// SIMATIC STEP 7 (V5.x) project Project
// CPU: CPU 315-2 DP
// station: Hardware
// station: SIMATIC 300(1)
// station: _S7H_BUSSYSTEM_CT
// station: P_ADR_BUS
// program: S7 Program(1)

SYMBOL_TABLE
"GLV"	DB 1	DB 1
"A_Sensors"	DB 2	DB 2
"DI"	DB 3	DB 3
"SensorsSettings"	DB 4	DB 4
"Valves"	DB 5	DB 5
"BD_Coils"	DB 6	DB 6
"KB1_1_Coils"	DB 7	DB 7
"KB1_2_Coils"	DB 8	DB 8
"KB2_Coils"	DB 9	DB 9
"PO1_1_Coils"	DB 10	DB 10
"PO1_2_Coils"	DB 11	DB 11
"GA1_1_Coils"	DB 12	DB 12
"GA1_2_Coils"	DB 13	DB 13
"GA2_1_Coils"	DB 14	DB 14
"GA2_2_Coils"	DB 15	DB 15
"BD_AI_1"	DB 16	DB 16
"KB1_1_AI_1"	DB 17	DB 17
"KB1_1_AI_2"	DB 18	DB 18
"KB1_1_AI_3"	DB 19	DB 19
"KB1_2_AI_1"	DB 20	DB 20
"KB1_2_AI_2"	DB 21	DB 21
"KB1_2_AI_3"	DB 22	DB 22
"KB2_AI_1"	DB 23	DB 23
"KB2_AI_2"	DB 24	DB 24
"KB2_AI_3"	DB 25	DB 25
"KB2_AI_4"	DB 26	DB 26
"PO1_1_AI"	DB 27	DB 27
"PO1_2_AI"	DB 28	DB 28
"GA1_1_AI_1"	DB 29	DB 29
"GA1_1_AI_2"	DB 30	DB 30
"GA1_2_AI_1"	DB 31	DB 31
"GA1_2_AI_2"	DB 32	DB 32
"GA2_1_AI_1"	DB 33	DB 33
"GA2_1_AI_2"	DB 34	DB 34
"KD1_1_AI"	DB 35	DB 35
"GA2_2_AI_1"	DB 36	DB 36
"GA2_2_AI_2"	DB 37	DB 37
"KD1_1_AI_2"	DB 38	DB 38
"KD1_1_AI_3"	DB 39	DB 39
"KD1_1_AI_4"	DB 40	DB 40
"KD1_1_AI_5"	DB 41	DB 41
"KD1_1_Coils"	DB 42	DB 42
"BD1_ARR_AI"	DB 43	DB 43
"BD_AI_2"	DB 44	DB 44
"BD_AI_3"	DB 45	DB 45
"BD_DO_1"	DB 46	DB 46
"BD_DO_2"	DB 47	DB 47
"GA1_1_DO"	DB 48	DB 48
"GA1_2_DO"	DB 49	DB 49
"GA2_1_DO"	DB 50	DB 50
"GA2_2_DO"	DB 51	DB 51
"BD_REAL"	DB 52	DB 52
"KB1_1_REAL"	DB 53	DB 53
"KB1_2_REAL"	DB 54	DB 54
"KB2_REAL"	DB 55	DB 55
"PO1_1_REAL"	DB 56	DB 56
"PO1_2_REAL"	DB 57	DB 57
"GA1_1_REAL"	DB 58	DB 58
"GA1_2_REAL"	DB 59	DB 59
"GA2_1_REAL"	DB 60	DB 60
"GA2_2_REAL"	DB 61	DB 61
"KD_REAL"	DB 62	DB 62
"ModbusVars"	DB 63	DB 63
"BD_Outputs_1"	DB 64	DB 64
"BD_Outputs_2"	DB 65	DB 65
"PO1_1_Outputs"	DB 66	DB 66
"PO1_2_Outputs"	DB 67	DB 67
"GA1_1_Outputs"	DB 68	DB 68
"GA1_2_Outputs"	DB 69	DB 69
"GA2_1_Outputs"	DB 97	DB 97
"GA2_2_Outputs"	DB 98	DB 98
"BD_OutputBytes_1"	DB 99	DB 99
"BD_OutputBytes_2"	DB 111	DB 111
"PO1_1_OutBytes"	DB 112	DB 112
"PO1_2_OutBytes"	DB 113	DB 113
"GA1_1_OutBytes"	DB 114	DB 114
"GA1_2_OutBytes"	DB 115	DB 115
"GA2_1_OutBytes"	DB 116	DB 116
"GA2_2_OutBytes"	DB 117	DB 117
"StartStop"	DB 118	DB 118
"StartStopBytes"	DB 119	DB 119
"KB2_AI_Bearer"	DB 128	DB 128
"KB2_AI_Vibration"	DB 129	DB 129
"ModbusAddresses"	DB 130	DB 130
"PO2_AI"	DB 131	DB 131
"PO2_Reals"	DB 132	DB 132
"PO2_AI2"	DB 133	DB 133
"DI_Bytes"	DB 134	DB 134
"PCV10_PID_Vars"	DB 135	DB 135
"PCV21_PID_Vars"	DB 136	DB 136
"PCV22_PID_Vars"	DB 137	DB 137
"PCV25_PID_Vars"	DB 138	DB 138
"ValvesVars"	DB 139	DB 139
"SensorsAlarmSettings"	DB 140	DB 140
"BD_MaxMin"	DB 141	DB 141
"GA1_1_MinMax"	DB 142	DB 142
"GA1_2_MinMax"	DB 143	DB 143
"GA2_1_MinMax"	DB 144	DB 144
"GA2_2_MinMax"	DB 145	DB 145
"KB1_1_MinMax"	DB 146	DB 146
"KB1_2_MinMax"	DB 147	DB 147
"KD2_ManMax"	DB 148	DB 148
"PO1_1_MaxMin"	DB 149	DB 149
"PO1_2_MinMax"	DB 150	DB 150
"ProcessSettings"	DB 151	DB 151
"ProcessVars"	DB 152	DB 152
"PrepareStartStop"	DB 153	DB 153
"PO2_Coils"	DB 154	DB 154
"PO2_MinMax"	DB 155	DB 155
"ZB1"	DB 777	FB 38
"ZB2"	DB 778	FB 38
"ZB3"	DB 779	FB 38
"ZB4"	DB 780	FB 38
"ValvesPrgDB"	DB 781	FB 39
"BD_GetReals"	FB 1	FB 1
"KB1_1_GetReals"	FB 2	FB 2
"KB1_2_GetReals"	FB 3	FB 3
"KB2_GetReals"	FB 4	FB 4
"PO1_1_GetReals"	FB 5	FB 5
"PO1_2_GetReals"	FB 6	FB 6
"P_RCV_RK"	FB 7	FB 7	// Receive Data / Provide Data
"P_SND_RK"	FB 8	FB 8	// Send Data / Fetch Data
"GA1_1_GetReal"	FB 9	FB 9
"MBMAREQ"	FB 10	FB 10	// MBMAREQ MODBUS MASTER REQUEST FUNCTION BLOCK
"GA1_2_GetReals"	FB 11	FB 11
"GA2_1_GetReals"	FB 12	FB 12
"GA2_2_GetReals"	FB 13	FB 13
"KD_GetReals"	FB 14	FB 14
"ModbusReal"	FB 15	FB 15
"ModbusCoils"	FB 16	FB 16
"ModbusOutputs"	FB 17	FB 17
"BD_GetOutputs"	FB 18	FB 18
"PO1_1_GetOutputs"	FB 19	FB 19
"PO1_2_GetOutputs"	FB 20	FB 20
"GA1_1_GetOutputs"	FB 21	FB 21
"GA1_2_GetOutputs"	FB 22	FB 22
"GA2_1_GetOutputs"	FB 23	FB 23
"GA2_2_GetOutputs"	FB 24	FB 24
"ModbusStartStop"	FB 25	FB 25
"GetStartStopBytes"	FB 26	FB 26
"GetAll"	FB 27	FB 27
"ModbusAll"	FB 28	FB 28
"InToVars"	FB 29	FB 29
"InToVarsST"	FB 30	FB 30
"PO2_GetReals"	FB 31	FB 31
"DI_ToVars"	FB 32	FB 32
"Valve_PID"	FB 33	FB 33
"fbPID"	FB 34	FB 34
"MBMA341"	FB 35	FB 35	// MBMA341 MODBUS MASTER COMMUNICATION FUNCTION BLOCK
"DERIVATIVE"	FB 36	FB 36
"INTEGRAL"	FB 37	FB 37
"DO_Valve"	FB 38	FB 38
"ValvesPrg"	FB 39	FB 39
"fbProcess_1"	FB 40	FB 40
"CONT_C"	FB 41	FB 41	// Continuous Control
"CONT_S"	FB 42	FB 42	// Step Control
"fbImpulsValve"	FB 43	FB 43
"fbImpulsValveSCL"	FB 44	FB 44
"prProcess"	FB 45	FB 45
"fbPO"	FB 46	FB 46
"fbKB"	FB 47	FB 47
"fbKZA"	FB 48	FB 48
"prDevices"	FB 49	FB 49
"GetCoils"	FB 50	FB 50
"LinTrafo"	FC 1	FC 1
"fnWordPack"	FC 2	FC 2
"fnBytesToReal"	FC 3	FC 3
"fnBytesToRealOneComma"	FC 4	FC 4
"fnBytesToRealPressure"	FC 5	FC 5
"fnBytesToRealTwoComas"	FC 6	FC 6
"StartStopByte"	FC 7	FC 7
"LinTrafoInt"	FC 8	FC 8
"ByteToByte"	FC 9	FC 9
"_DI_XL1_QL3"	I 0.0	BOOL
"_DI_XL2_QL3"	I 0.1	BOOL
"_DI_Q3_Bad"	I 0.2	BOOL
"_DI_AB1_Working"	I 0.3	BOOL
"_DI_Kb_1_1_Working"	I 0.4	BOOL
"_DI_Kb_1_1_Alm"	I 0.5	BOOL
"_DI_Kb_1_2_Working"	I 0.6	BOOL
"_DI_Kb_1_2_Alm"	I 0.7	BOOL
"_DI_Kb_2_Working"	I 1.0	BOOL
"_DI_Kb_2_Alm"	I 1.1	BOOL
"_DI_Kd_1_Working"	I 1.2	BOOL
"_DI_Kd_1_Alm"	I 1.3	BOOL
"_DI_ZB_1_Opn"	I 1.4	BOOL
"_DI_ZB_1_Cls"	I 1.5	BOOL
"_DI_ZB_1_Local"	I 1.6	BOOL
"_DI_ZB_1_Alm"	I 1.7	BOOL
"_DI_ZB_2_Opn"	I 2.0	BOOL
"_DI_ZB_2_Cls"	I 2.1	BOOL
"_DI_ZB_2_Local"	I 2.2	BOOL
"_DI_ZB_2_Alm"	I 2.3	BOOL
"_DI_ZB_3_Opn"	I 2.4	BOOL
"_DI_ZB_3_Cls"	I 2.5	BOOL
"_DI_ZB_3_Local"	I 2.6	BOOL
"_DI_ZB_3_Alm"	I 2.7	BOOL
"_DI_EUV_001_Opn"	I 3.0	BOOL
"_DI_EUV_001_Cls"	I 3.1	BOOL
"_DI_EUV_001_Local"	I 3.2	BOOL
"_DI_EUV_001_Alm"	I 3.3	BOOL
"_DI_EUV_002_Opn"	I 3.4	BOOL
"_DI_EUV_002_Cls"	I 3.5	BOOL
"_DI_EUV_002_Local"	I 3.6	BOOL
"_DI_EUV_002_Alm"	I 3.7	BOOL
"_DI_EUV_003_Opn"	I 4.0	BOOL
"_DI_EUV_003_Cls"	I 4.1	BOOL
"_DI_EUV_003_Local"	I 4.2	BOOL
"_DI_EUV_003_Alm"	I 4.3	BOOL
"QSA_19_1_1"	I 4.4	BOOL
"QSA_23_1_1"	I 4.5	BOOL
"QSA_19_1_2"	I 4.6	BOOL
"QSA_23_1_2"	I 4.7	BOOL
"QSA_19_1_3"	I 5.0	BOOL
"QSA_23_1_3"	I 5.1	BOOL
"QSA_19_1_4"	I 5.2	BOOL
"QSA_23_1_4"	I 5.3	BOOL
"QSA_19_1_5"	I 5.4	BOOL
"QSA_23_1_5"	I 5.5	BOOL
"Q3_BAD"	I 5.6	BOOL
"AB_1_Alm"	I 5.7	BOOL
"AB_2_Working"	I 6.0	BOOL
"AB_2_Alm"	I 6.1	BOOL
"AB_3_Working"	I 6.2	BOOL
"AB_3_Alm"	I 6.3	BOOL
"AB_4_Working"	I 6.4	BOOL
"AB_4_Alm"	I 6.5	BOOL
"P2_Alm"	I 6.6	BOOL
"P2_Working"	I 6.7	BOOL
"P3_Alm"	I 7.0	BOOL
"P3_Working"	I 7.1	BOOL
"IBP_1_Working"	I 7.2	BOOL
"IBP_1_Alm"	I 7.3	BOOL
"IBP_1_Bypas"	I 7.4	BOOL
"IBP_2_Working"	I 7.5	BOOL
"IBP_2_Alm"	I 7.6	BOOL
"IBP_2_Bypas"	I 7.7	BOOL
"_DI_ZB_4_Opn"	I 8.0	BOOL
"_DI_ZB_4_Cls"	I 8.1	BOOL
"_DI_ZB_4_Local"	I 8.2	BOOL
"_DI_ZB_4_Alm"	I 8.3	BOOL
"_KB_1_1_1PIR7"	IW 256	WORD
"_KB_1_2_2PIR7"	IW 258	WORD
"_1PIR6"	IW 260	WORD
"_KZA_1_2_2PIR6"	IW 262	WORD
"_KB_2_PIR8"	IW 264	WORD
"_1PIR20"	IW 266	WORD
"_2PIR20"	IW 268	WORD
"_TIR10"	IW 270	WORD
"_FIR10"	IW 272	WORD
"_PIR5"	IW 274	WORD
"_FIR5"	IW 276	WORD
"_PIRC21"	IW 278	WORD
"_1PIR27"	IW 280	WORD
"_QIRAH3"	IW 282	WORD
"_2PIR27"	IW 284	WORD
"_PIR4"	IW 286	WORD
"_FIR_4"	IW 288	WORD
"_PIRC22"	IW 290	WORD
"_PIRC23"	IW 292	WORD
"_PIRC24"	IW 294	WORD
"_PIRC25"	IW 296	WORD
"_FIR_25"	IW 298	WORD
"_1PIRC26"	IW 300	WORD
"_2PIRC26"	IW 302	WORD
"_C10"	IW 304	WORD
"_TIR5"	IW 306	WORD
"_TIR4"	IW 308	WORD
"_TIR25"	IW 310	WORD
"_AIR1"	IW 312	WORD
"_QIRAH4Q4"	IW 314	WORD
"CYC_INT5"	OB 35	OB 35	// Cyclic Interrupt 5
"_DO_HS1Q1_Acknow"	Q 0.0	BOOL
"_DO_HS1Q1_Check"	Q 0.1	BOOL
"_DO_KB_1_1_Stop"	Q 0.2	BOOL
"_DO_KB_1_1_Start"	Q 0.3	BOOL
"_DO_KB_1_2_Stop"	Q 0.4	BOOL
"_DO_KB_1_2_Start"	Q 0.5	BOOL
"_DO_KB_2_Stop"	Q 0.6	BOOL
"_DO_KB_2_Start"	Q 0.7	BOOL
"_DO_KD_1_Start"	Q 1.0	BOOL
"_DO_KD_1_Stop"	Q 1.1	BOOL
"_DO_ZB_1_CmdOpn"	Q 1.2	BOOL
"_DO_ZB_1_CmdCls"	Q 1.3	BOOL
"_DO_ZB_1_CmdStop"	Q 1.4	BOOL
"_DO_ZB_2_CmdOpn"	Q 1.5	BOOL
"_DO_ZB_2_CmdCls"	Q 1.6	BOOL
"_DO_ZB_2_CmdStop"	Q 1.7	BOOL
"_DO_ZB_3_CmdOpn"	Q 2.0	BOOL
"_DO_ZB_3_CmdCls"	Q 2.1	BOOL
"_DO_ZB_3_CmdStop"	Q 2.2	BOOL
"_DO_AlnVent"	Q 2.3	BOOL
"_DO_ZB_4_CmdOpn"	Q 2.4	BOOL
"_DO_ZB_4_CmdCls"	Q 2.5	BOOL
"_DO_ZB_4_CmdStop"	Q 2.6	BOOL
"_AO_N_Set_PCV10"	QW 256	WORD
"_AO_N_Set_PCV21"	QW 258	WORD
"_AO_Air_Set_PCV22"	QW 260	WORD
"_AO_Air_Set_PCV25"	QW 262	WORD
"RDREC"	SFB 52	SFB 52	// Read a Process Data Record
"WRREC"	SFB 53	SFB 53	// Write a Process Data Record
"DI_Vars"	VAT 1	
"DO_Vars"	VAT 2	
"AI_Vars"	VAT 3	
"AO_Vars"	VAT 4	
END_SYMBOL_TABLE

FUNCTION_BLOCK "BD_GetReals"	// FB 1
VERSION : 0.1
BEGIN
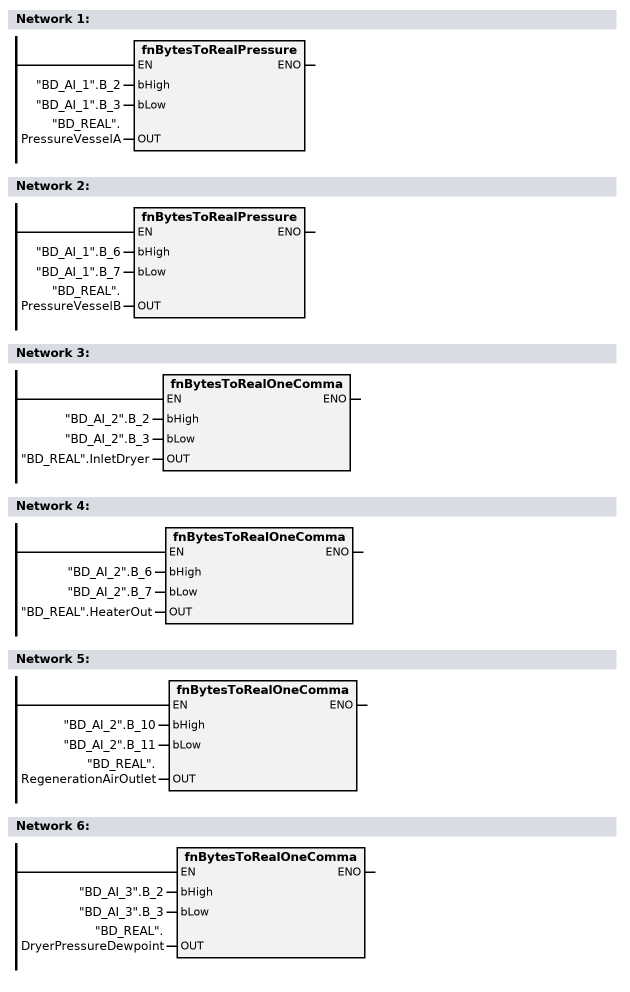
NETWORK
TITLE =
      CALL  "fnBytesToRealPressure" (
           bHigh                    := "BD_AI_1".B_2,
           bLow                     := "BD_AI_1".B_3,
           OUT                      := "BD_REAL".PressureVesselA);
      NOP   0;
NETWORK
TITLE =
      CALL  "fnBytesToRealPressure" (
           bHigh                    := "BD_AI_1".B_6,
           bLow                     := "BD_AI_1".B_7,
           OUT                      := "BD_REAL".PressureVesselB);
      NOP   0;
NETWORK
TITLE =
      CALL  "fnBytesToRealOneComma" (
           bHigh                    := "BD_AI_2".B_2,
           bLow                     := "BD_AI_2".B_3,
           OUT                      := "BD_REAL".InletDryer);
      NOP   0;
NETWORK
TITLE =
      CALL  "fnBytesToRealOneComma" (
           bHigh                    := "BD_AI_2".B_6,
           bLow                     := "BD_AI_2".B_7,
           OUT                      := "BD_REAL".HeaterOut);
      NOP   0;
NETWORK
TITLE =
      CALL  "fnBytesToRealOneComma" (
           bHigh                    := "BD_AI_2".B_10,
           bLow                     := "BD_AI_2".B_11,
           OUT                      := "BD_REAL".RegenerationAirOutlet);
      NOP   0;
NETWORK
TITLE =
      CALL  "fnBytesToRealOneComma" (
           bHigh                    := "BD_AI_3".B_2,
           bLow                     := "BD_AI_3".B_3,
           OUT                      := "BD_REAL".DryerPressureDewpoint);
      NOP   0;
END_FUNCTION_BLOCK

FUNCTION_BLOCK "KB1_1_GetReals"	// FB 2
VERSION : 0.1
BEGIN
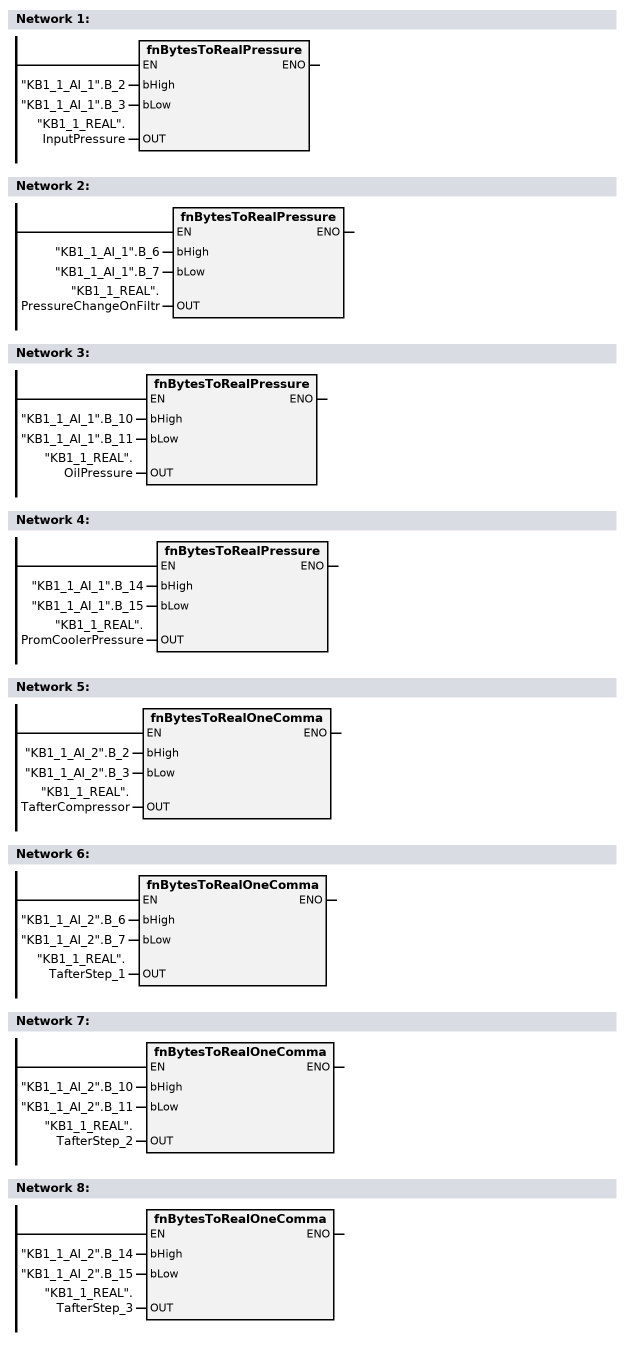
NETWORK
TITLE =
      CALL  "fnBytesToRealPressure" (
           bHigh                    := "KB1_1_AI_1".B_2,
           bLow                     := "KB1_1_AI_1".B_3,
           OUT                      := "KB1_1_REAL".InputPressure);
      NOP   0;
NETWORK
TITLE =
      CALL  "fnBytesToRealPressure" (
           bHigh                    := "KB1_1_AI_1".B_6,
           bLow                     := "KB1_1_AI_1".B_7,
           OUT                      := "KB1_1_REAL".PressureChangeOnFiltr);
      NOP   0;
NETWORK
TITLE =
      CALL  "fnBytesToRealPressure" (
           bHigh                    := "KB1_1_AI_1".B_10,
           bLow                     := "KB1_1_AI_1".B_11,
           OUT                      := "KB1_1_REAL".OilPressure);
      NOP   0;
NETWORK
TITLE =
      CALL  "fnBytesToRealPressure" (
           bHigh                    := "KB1_1_AI_1".B_14,
           bLow                     := "KB1_1_AI_1".B_15,
           OUT                      := "KB1_1_REAL".PromCoolerPressure);
      NOP   0;
NETWORK
TITLE =
      CALL  "fnBytesToRealOneComma" (
           bHigh                    := "KB1_1_AI_2".B_2,
           bLow                     := "KB1_1_AI_2".B_3,
           OUT                      := "KB1_1_REAL".TafterCompressor);
      NOP   0;
NETWORK
TITLE =
      CALL  "fnBytesToRealOneComma" (
           bHigh                    := "KB1_1_AI_2".B_6,
           bLow                     := "KB1_1_AI_2".B_7,
           OUT                      := "KB1_1_REAL".TafterStep_1);
      NOP   0;
NETWORK
TITLE =
      CALL  "fnBytesToRealOneComma" (
           bHigh                    := "KB1_1_AI_2".B_10,
           bLow                     := "KB1_1_AI_2".B_11,
           OUT                      := "KB1_1_REAL".TafterStep_2);
      NOP   0;
NETWORK
TITLE =
      CALL  "fnBytesToRealOneComma" (
           bHigh                    := "KB1_1_AI_2".B_14,
           bLow                     := "KB1_1_AI_2".B_15,
           OUT                      := "KB1_1_REAL".TafterStep_3);
      NOP   0;
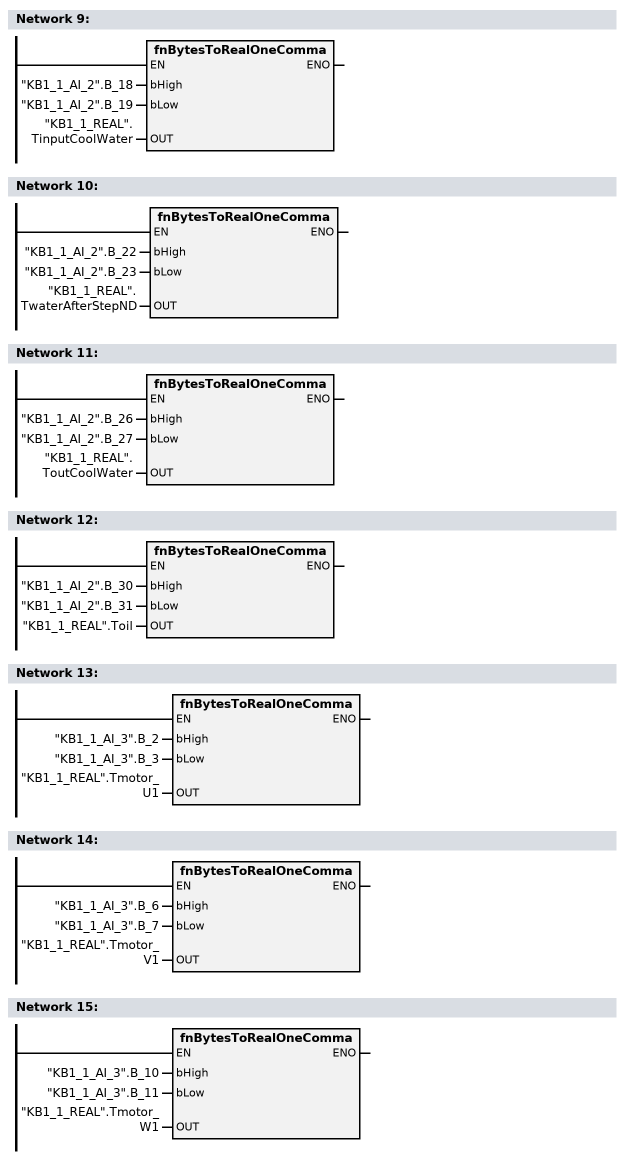
NETWORK
TITLE =
      CALL  "fnBytesToRealOneComma" (
           bHigh                    := "KB1_1_AI_2".B_18,
           bLow                     := "KB1_1_AI_2".B_19,
           OUT                      := "KB1_1_REAL".TinputCoolWater);
      NOP   0;
NETWORK
TITLE =
      CALL  "fnBytesToRealOneComma" (
           bHigh                    := "KB1_1_AI_2".B_22,
           bLow                     := "KB1_1_AI_2".B_23,
           OUT                      := "KB1_1_REAL".TwaterAfterStepND);
      NOP   0;
NETWORK
TITLE =
      CALL  "fnBytesToRealOneComma" (
           bHigh                    := "KB1_1_AI_2".B_26,
           bLow                     := "KB1_1_AI_2".B_27,
           OUT                      := "KB1_1_REAL".ToutCoolWater);
      NOP   0;
NETWORK
TITLE =
      CALL  "fnBytesToRealOneComma" (
           bHigh                    := "KB1_1_AI_2".B_30,
           bLow                     := "KB1_1_AI_2".B_31,
           OUT                      := "KB1_1_REAL".Toil);
      NOP   0;
NETWORK
TITLE =
      CALL  "fnBytesToRealOneComma" (
           bHigh                    := "KB1_1_AI_3".B_2,
           bLow                     := "KB1_1_AI_3".B_3,
           OUT                      := "KB1_1_REAL".Tmotor_U1);
      NOP   0;
NETWORK
TITLE =
      CALL  "fnBytesToRealOneComma" (
           bHigh                    := "KB1_1_AI_3".B_6,
           bLow                     := "KB1_1_AI_3".B_7,
           OUT                      := "KB1_1_REAL".Tmotor_V1);
      NOP   0;
NETWORK
TITLE =
      CALL  "fnBytesToRealOneComma" (
           bHigh                    := "KB1_1_AI_3".B_10,
           bLow                     := "KB1_1_AI_3".B_11,
           OUT                      := "KB1_1_REAL".Tmotor_W1);
      NOP   0;
END_FUNCTION_BLOCK

FUNCTION_BLOCK "KB1_2_GetReals"	// FB 3
VERSION : 0.1
BEGIN
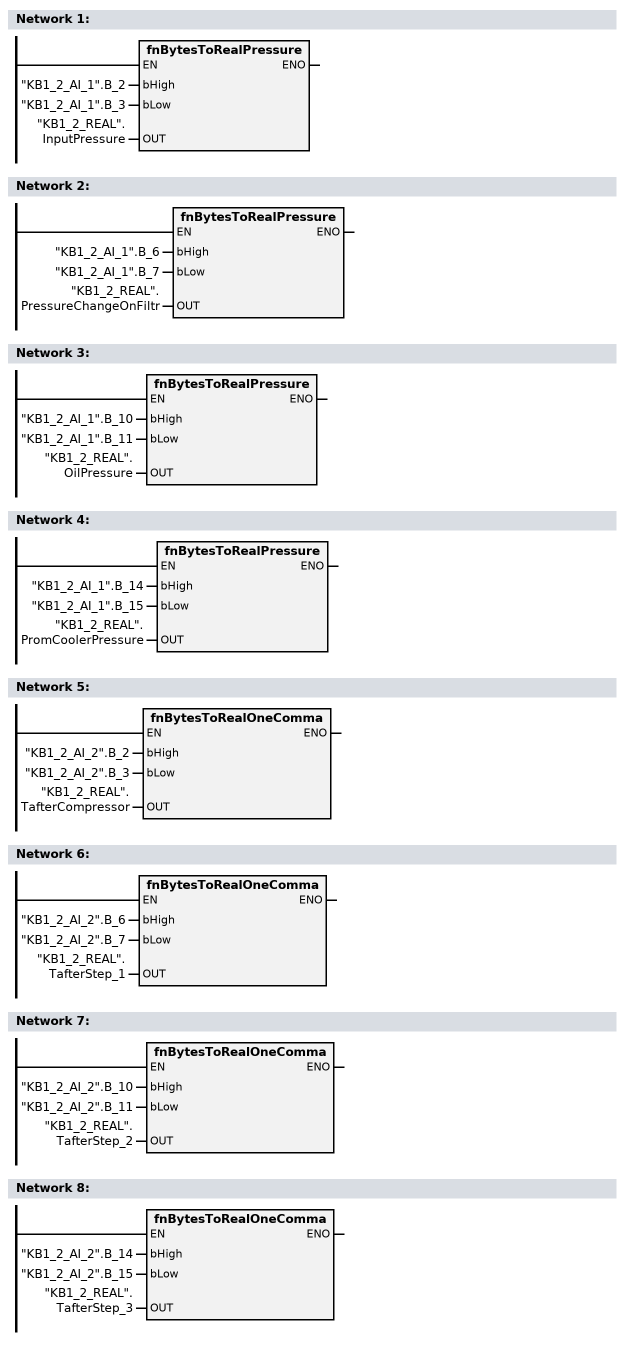
NETWORK
TITLE =
      CALL  "fnBytesToRealPressure" (
           bHigh                    := "KB1_2_AI_1".B_2,
           bLow                     := "KB1_2_AI_1".B_3,
           OUT                      := "KB1_2_REAL".InputPressure);
      NOP   0;
NETWORK
TITLE =
      CALL  "fnBytesToRealPressure" (
           bHigh                    := "KB1_2_AI_1".B_6,
           bLow                     := "KB1_2_AI_1".B_7,
           OUT                      := "KB1_2_REAL".PressureChangeOnFiltr);
      NOP   0;
NETWORK
TITLE =
      CALL  "fnBytesToRealPressure" (
           bHigh                    := "KB1_2_AI_1".B_10,
           bLow                     := "KB1_2_AI_1".B_11,
           OUT                      := "KB1_2_REAL".OilPressure);
      NOP   0;
NETWORK
TITLE =
      CALL  "fnBytesToRealPressure" (
           bHigh                    := "KB1_2_AI_1".B_14,
           bLow                     := "KB1_2_AI_1".B_15,
           OUT                      := "KB1_2_REAL".PromCoolerPressure);
      NOP   0;
NETWORK
TITLE =
      CALL  "fnBytesToRealOneComma" (
           bHigh                    := "KB1_2_AI_2".B_2,
           bLow                     := "KB1_2_AI_2".B_3,
           OUT                      := "KB1_2_REAL".TafterCompressor);
      NOP   0;
NETWORK
TITLE =
      CALL  "fnBytesToRealOneComma" (
           bHigh                    := "KB1_2_AI_2".B_6,
           bLow                     := "KB1_2_AI_2".B_7,
           OUT                      := "KB1_2_REAL".TafterStep_1);
      NOP   0;
NETWORK
TITLE =
      CALL  "fnBytesToRealOneComma" (
           bHigh                    := "KB1_2_AI_2".B_10,
           bLow                     := "KB1_2_AI_2".B_11,
           OUT                      := "KB1_2_REAL".TafterStep_2);
      NOP   0;
NETWORK
TITLE =
      CALL  "fnBytesToRealOneComma" (
           bHigh                    := "KB1_2_AI_2".B_14,
           bLow                     := "KB1_2_AI_2".B_15,
           OUT                      := "KB1_2_REAL".TafterStep_3);
      NOP   0;
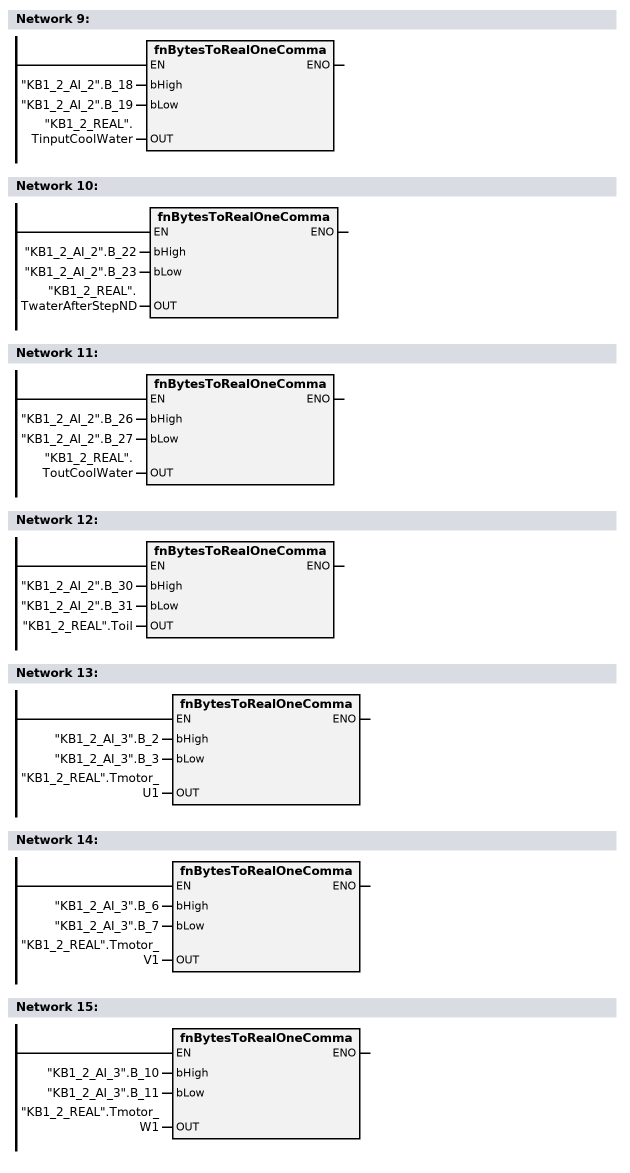
NETWORK
TITLE =
      CALL  "fnBytesToRealOneComma" (
           bHigh                    := "KB1_2_AI_2".B_18,
           bLow                     := "KB1_2_AI_2".B_19,
           OUT                      := "KB1_2_REAL".TinputCoolWater);
      NOP   0;
NETWORK
TITLE =
      CALL  "fnBytesToRealOneComma" (
           bHigh                    := "KB1_2_AI_2".B_22,
           bLow                     := "KB1_2_AI_2".B_23,
           OUT                      := "KB1_2_REAL".TwaterAfterStepND);
      NOP   0;
NETWORK
TITLE =
      CALL  "fnBytesToRealOneComma" (
           bHigh                    := "KB1_2_AI_2".B_26,
           bLow                     := "KB1_2_AI_2".B_27,
           OUT                      := "KB1_2_REAL".ToutCoolWater);
      NOP   0;
NETWORK
TITLE =
      CALL  "fnBytesToRealOneComma" (
           bHigh                    := "KB1_2_AI_2".B_30,
           bLow                     := "KB1_2_AI_2".B_31,
           OUT                      := "KB1_2_REAL".Toil);
      NOP   0;
NETWORK
TITLE =
      CALL  "fnBytesToRealOneComma" (
           bHigh                    := "KB1_2_AI_3".B_2,
           bLow                     := "KB1_2_AI_3".B_3,
           OUT                      := "KB1_2_REAL".Tmotor_U1);
      NOP   0;
NETWORK
TITLE =
      CALL  "fnBytesToRealOneComma" (
           bHigh                    := "KB1_2_AI_3".B_6,
           bLow                     := "KB1_2_AI_3".B_7,
           OUT                      := "KB1_2_REAL".Tmotor_V1);
      NOP   0;
NETWORK
TITLE =
      CALL  "fnBytesToRealOneComma" (
           bHigh                    := "KB1_2_AI_3".B_10,
           bLow                     := "KB1_2_AI_3".B_11,
           OUT                      := "KB1_2_REAL".Tmotor_W1);
      NOP   0;
END_FUNCTION_BLOCK

FUNCTION_BLOCK "KB2_GetReals"	// FB 4
VERSION : 0.1
BEGIN
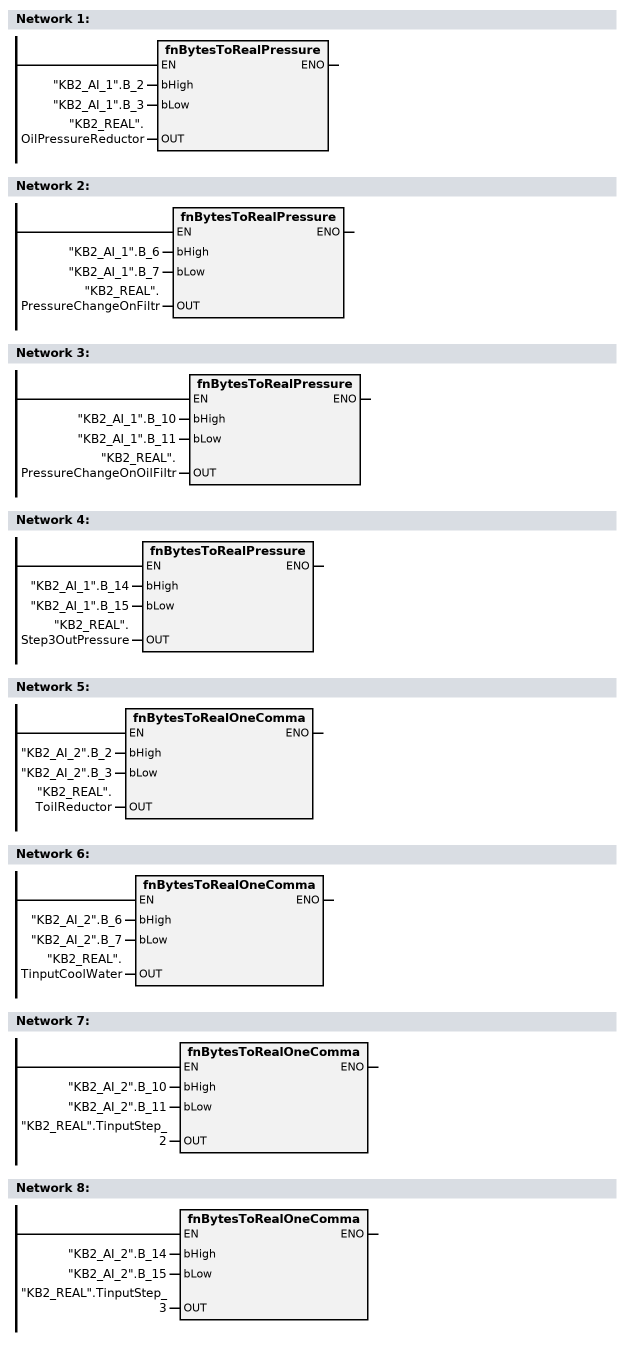
NETWORK
TITLE =
      CALL  "fnBytesToRealPressure" (
           bHigh                    := "KB2_AI_1".B_2,
           bLow                     := "KB2_AI_1".B_3,
           OUT                      := "KB2_REAL".OilPressureReductor);
      NOP   0;
NETWORK
TITLE =
      CALL  "fnBytesToRealPressure" (
           bHigh                    := "KB2_AI_1".B_6,
           bLow                     := "KB2_AI_1".B_7,
           OUT                      := "KB2_REAL".PressureChangeOnFiltr);
      NOP   0;
NETWORK
TITLE =
      CALL  "fnBytesToRealPressure" (
           bHigh                    := "KB2_AI_1".B_10,
           bLow                     := "KB2_AI_1".B_11,
           OUT                      := "KB2_REAL".PressureChangeOnOilFiltr);
      NOP   0;
NETWORK
TITLE =
      CALL  "fnBytesToRealPressure" (
           bHigh                    := "KB2_AI_1".B_14,
           bLow                     := "KB2_AI_1".B_15,
           OUT                      := "KB2_REAL".Step3OutPressure);
      NOP   0;
NETWORK
TITLE =
      CALL  "fnBytesToRealOneComma" (
           bHigh                    := "KB2_AI_2".B_2,
           bLow                     := "KB2_AI_2".B_3,
           OUT                      := "KB2_REAL".ToilReductor);
      NOP   0;
NETWORK
TITLE =
      CALL  "fnBytesToRealOneComma" (
           bHigh                    := "KB2_AI_2".B_6,
           bLow                     := "KB2_AI_2".B_7,
           OUT                      := "KB2_REAL".TinputCoolWater);
      NOP   0;
NETWORK
TITLE =
      CALL  "fnBytesToRealOneComma" (
           bHigh                    := "KB2_AI_2".B_10,
           bLow                     := "KB2_AI_2".B_11,
           OUT                      := "KB2_REAL".TinputStep_2);
      NOP   0;
NETWORK
TITLE =
      CALL  "fnBytesToRealOneComma" (
           bHigh                    := "KB2_AI_2".B_14,
           bLow                     := "KB2_AI_2".B_15,
           OUT                      := "KB2_REAL".TinputStep_3);
      NOP   0;
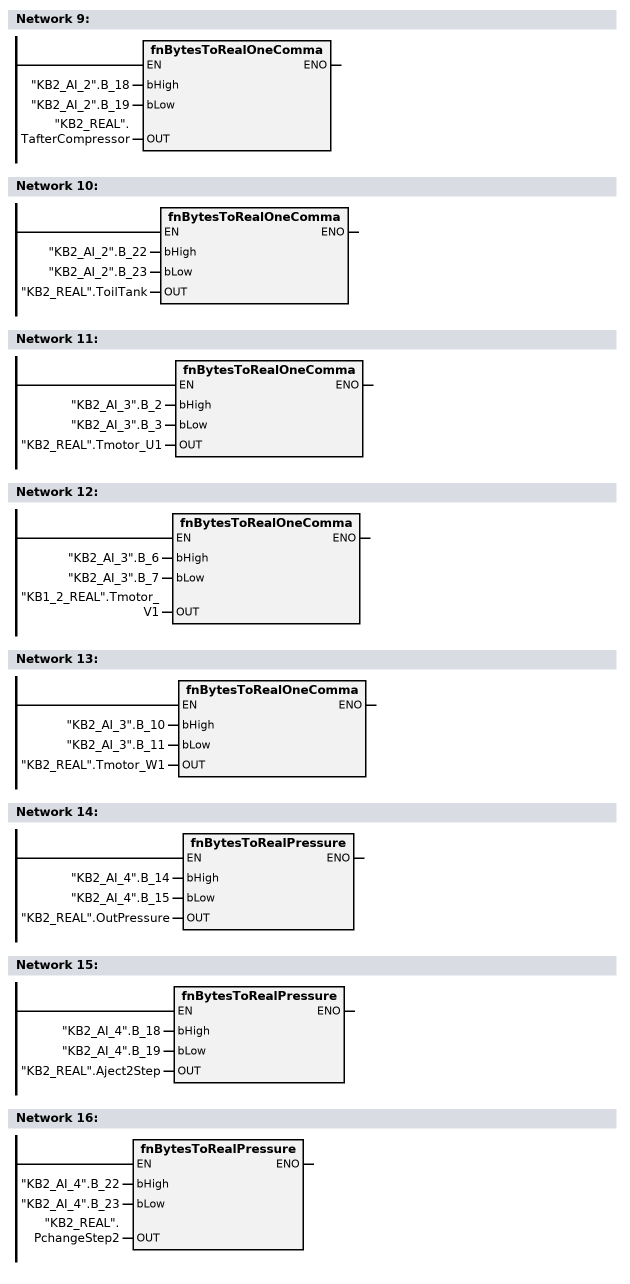
NETWORK
TITLE =
      CALL  "fnBytesToRealOneComma" (
           bHigh                    := "KB2_AI_2".B_18,
           bLow                     := "KB2_AI_2".B_19,
           OUT                      := "KB2_REAL".TafterCompressor);
      NOP   0;
NETWORK
TITLE =
      CALL  "fnBytesToRealOneComma" (
           bHigh                    := "KB2_AI_2".B_22,
           bLow                     := "KB2_AI_2".B_23,
           OUT                      := "KB2_REAL".ToilTank);
      NOP   0;
NETWORK
TITLE =
      CALL  "fnBytesToRealOneComma" (
           bHigh                    := "KB2_AI_3".B_2,
           bLow                     := "KB2_AI_3".B_3,
           OUT                      := "KB2_REAL".Tmotor_U1);
      NOP   0;
NETWORK
TITLE =
      CALL  "fnBytesToRealOneComma" (
           bHigh                    := "KB2_AI_3".B_6,
           bLow                     := "KB2_AI_3".B_7,
           OUT                      := "KB1_2_REAL".Tmotor_V1);
      NOP   0;
NETWORK
TITLE =
      CALL  "fnBytesToRealOneComma" (
           bHigh                    := "KB2_AI_3".B_10,
           bLow                     := "KB2_AI_3".B_11,
           OUT                      := "KB2_REAL".Tmotor_W1);
      NOP   0;
NETWORK
TITLE =
      CALL  "fnBytesToRealPressure" (
           bHigh                    := "KB2_AI_4".B_14,
           bLow                     := "KB2_AI_4".B_15,
           OUT                      := "KB2_REAL".OutPressure);
      NOP   0;
NETWORK
TITLE =
      CALL  "fnBytesToRealPressure" (
           bHigh                    := "KB2_AI_4".B_18,
           bLow                     := "KB2_AI_4".B_19,
           OUT                      := "KB2_REAL".Aject2Step);
      NOP   0;
NETWORK
TITLE =
      CALL  "fnBytesToRealPressure" (
           bHigh                    := "KB2_AI_4".B_22,
           bLow                     := "KB2_AI_4".B_23,
           OUT                      := "KB2_REAL".PchangeStep2);
      NOP   0;
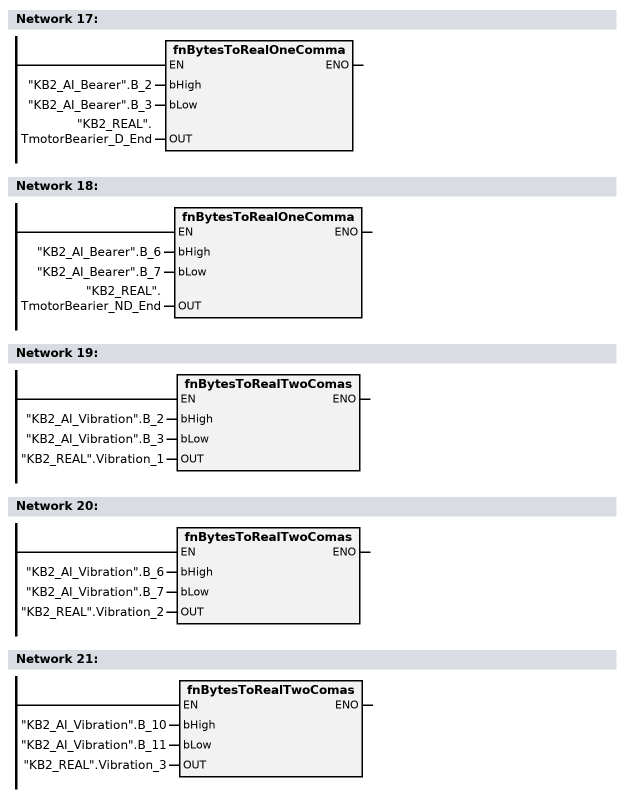
NETWORK
TITLE =
      CALL  "fnBytesToRealOneComma" (
           bHigh                    := "KB2_AI_Bearer".B_2,
           bLow                     := "KB2_AI_Bearer".B_3,
           OUT                      := "KB2_REAL".TmotorBearier_D_End);
      NOP   0;
NETWORK
TITLE =
      CALL  "fnBytesToRealOneComma" (
           bHigh                    := "KB2_AI_Bearer".B_6,
           bLow                     := "KB2_AI_Bearer".B_7,
           OUT                      := "KB2_REAL".TmotorBearier_ND_End);
      NOP   0;
NETWORK
TITLE =
      CALL  "fnBytesToRealTwoComas" (
           bHigh                    := "KB2_AI_Vibration".B_2,
           bLow                     := "KB2_AI_Vibration".B_3,
           OUT                      := "KB2_REAL".Vibration_1);
      NOP   0;
NETWORK
TITLE =
      CALL  "fnBytesToRealTwoComas" (
           bHigh                    := "KB2_AI_Vibration".B_6,
           bLow                     := "KB2_AI_Vibration".B_7,
           OUT                      := "KB2_REAL".Vibration_2);
      NOP   0;
NETWORK
TITLE =
      CALL  "fnBytesToRealTwoComas" (
           bHigh                    := "KB2_AI_Vibration".B_10,
           bLow                     := "KB2_AI_Vibration".B_11,
           OUT                      := "KB2_REAL".Vibration_3);
      NOP   0;
END_FUNCTION_BLOCK

FUNCTION_BLOCK "PO1_1_GetReals"	// FB 5
VERSION : 0.1
BEGIN
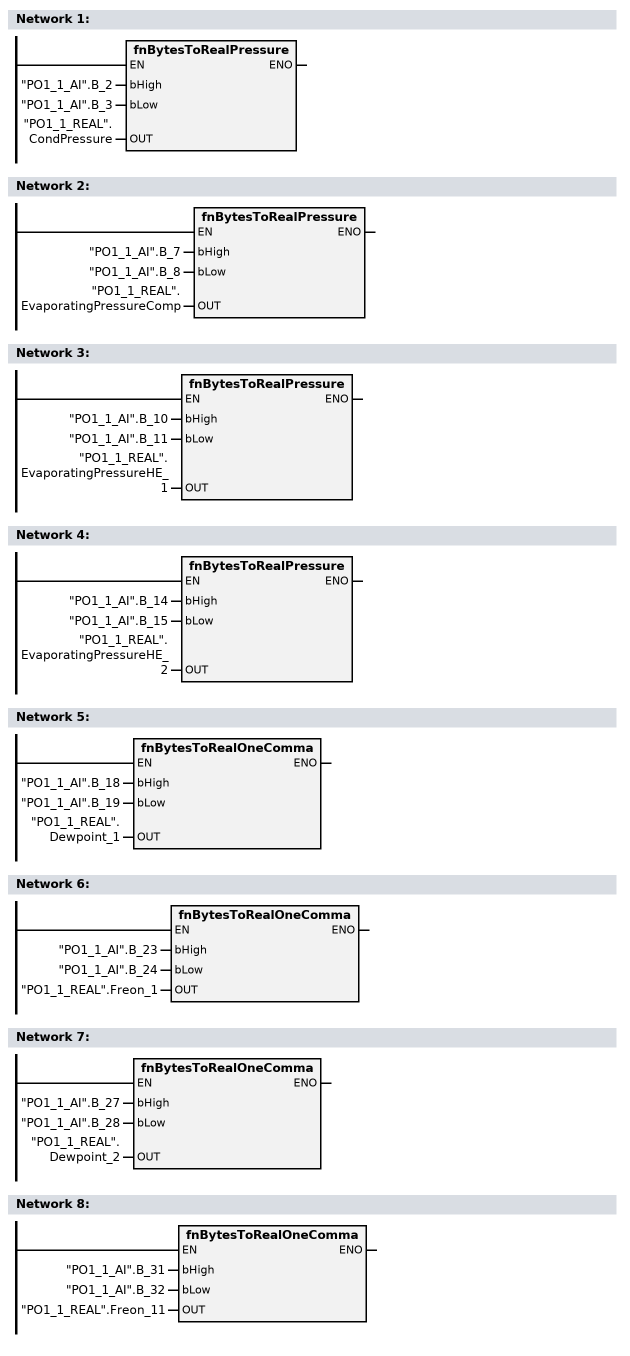
NETWORK
TITLE =
      CALL  "fnBytesToRealPressure" (
           bHigh                    := "PO1_1_AI".B_2,
           bLow                     := "PO1_1_AI".B_3,
           OUT                      := "PO1_1_REAL".CondPressure);
      NOP   0;
NETWORK
TITLE =
      CALL  "fnBytesToRealPressure" (
           bHigh                    := "PO1_1_AI".B_7,
           bLow                     := "PO1_1_AI".B_8,
           OUT                      := "PO1_1_REAL".EvaporatingPressureComp);
      NOP   0;
NETWORK
TITLE =
      CALL  "fnBytesToRealPressure" (
           bHigh                    := "PO1_1_AI".B_10,
           bLow                     := "PO1_1_AI".B_11,
           OUT                      := "PO1_1_REAL".EvaporatingPressureHE_1);
      NOP   0;
NETWORK
TITLE =
      CALL  "fnBytesToRealPressure" (
           bHigh                    := "PO1_1_AI".B_14,
           bLow                     := "PO1_1_AI".B_15,
           OUT                      := "PO1_1_REAL".EvaporatingPressureHE_2);
      NOP   0;
NETWORK
TITLE =
      CALL  "fnBytesToRealOneComma" (
           bHigh                    := "PO1_1_AI".B_18,
           bLow                     := "PO1_1_AI".B_19,
           OUT                      := "PO1_1_REAL".Dewpoint_1);
      NOP   0;
NETWORK
TITLE =
      CALL  "fnBytesToRealOneComma" (
           bHigh                    := "PO1_1_AI".B_23,
           bLow                     := "PO1_1_AI".B_24,
           OUT                      := "PO1_1_REAL".Freon_1);
      NOP   0;
NETWORK
TITLE =
      CALL  "fnBytesToRealOneComma" (
           bHigh                    := "PO1_1_AI".B_27,
           bLow                     := "PO1_1_AI".B_28,
           OUT                      := "PO1_1_REAL".Dewpoint_2);
      NOP   0;
NETWORK
TITLE =
      CALL  "fnBytesToRealOneComma" (
           bHigh                    := "PO1_1_AI".B_31,
           bLow                     := "PO1_1_AI".B_32,
           OUT                      := "PO1_1_REAL".Freon_11);
      NOP   0;
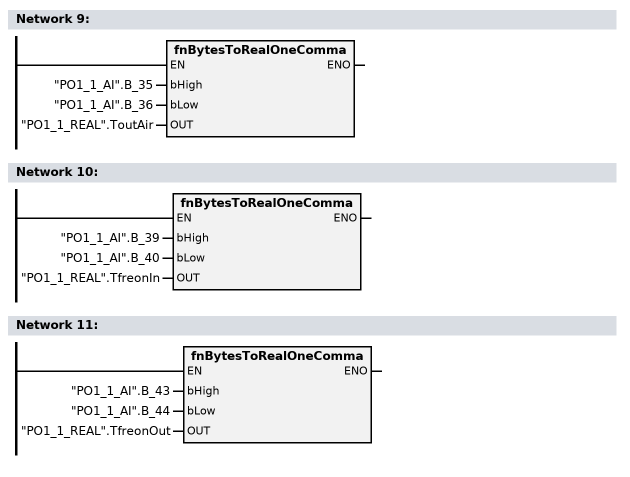
NETWORK
TITLE =
      CALL  "fnBytesToRealOneComma" (
           bHigh                    := "PO1_1_AI".B_35,
           bLow                     := "PO1_1_AI".B_36,
           OUT                      := "PO1_1_REAL".ToutAir);
      NOP   0;
NETWORK
TITLE =
      CALL  "fnBytesToRealOneComma" (
           bHigh                    := "PO1_1_AI".B_39,
           bLow                     := "PO1_1_AI".B_40,
           OUT                      := "PO1_1_REAL".TfreonIn);
      NOP   0;
NETWORK
TITLE =
      CALL  "fnBytesToRealOneComma" (
           bHigh                    := "PO1_1_AI".B_43,
           bLow                     := "PO1_1_AI".B_44,
           OUT                      := "PO1_1_REAL".TfreonOut);
      NOP   0;
END_FUNCTION_BLOCK

FUNCTION_BLOCK "PO1_2_GetReals"	// FB 6
VERSION : 0.1
BEGIN
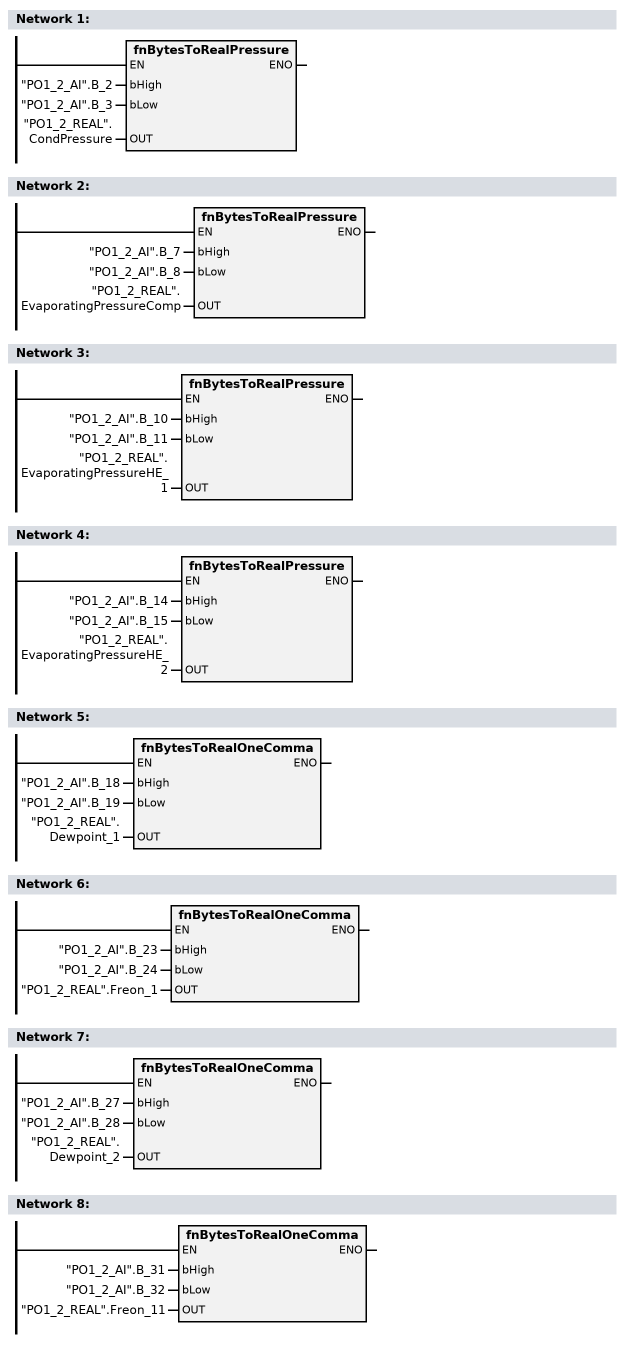
NETWORK
TITLE =
      CALL  "fnBytesToRealPressure" (
           bHigh                    := "PO1_2_AI".B_2,
           bLow                     := "PO1_2_AI".B_3,
           OUT                      := "PO1_2_REAL".CondPressure);
      NOP   0;
NETWORK
TITLE =
      CALL  "fnBytesToRealPressure" (
           bHigh                    := "PO1_2_AI".B_7,
           bLow                     := "PO1_2_AI".B_8,
           OUT                      := "PO1_2_REAL".EvaporatingPressureComp);
      NOP   0;
NETWORK
TITLE =
      CALL  "fnBytesToRealPressure" (
           bHigh                    := "PO1_2_AI".B_10,
           bLow                     := "PO1_2_AI".B_11,
           OUT                      := "PO1_2_REAL".EvaporatingPressureHE_1);
      NOP   0;
NETWORK
TITLE =
      CALL  "fnBytesToRealPressure" (
           bHigh                    := "PO1_2_AI".B_14,
           bLow                     := "PO1_2_AI".B_15,
           OUT                      := "PO1_2_REAL".EvaporatingPressureHE_2);
      NOP   0;
NETWORK
TITLE =
      CALL  "fnBytesToRealOneComma" (
           bHigh                    := "PO1_2_AI".B_18,
           bLow                     := "PO1_2_AI".B_19,
           OUT                      := "PO1_2_REAL".Dewpoint_1);
      NOP   0;
NETWORK
TITLE =
      CALL  "fnBytesToRealOneComma" (
           bHigh                    := "PO1_2_AI".B_23,
           bLow                     := "PO1_2_AI".B_24,
           OUT                      := "PO1_2_REAL".Freon_1);
      NOP   0;
NETWORK
TITLE =
      CALL  "fnBytesToRealOneComma" (
           bHigh                    := "PO1_2_AI".B_27,
           bLow                     := "PO1_2_AI".B_28,
           OUT                      := "PO1_2_REAL".Dewpoint_2);
      NOP   0;
NETWORK
TITLE =
      CALL  "fnBytesToRealOneComma" (
           bHigh                    := "PO1_2_AI".B_31,
           bLow                     := "PO1_2_AI".B_32,
           OUT                      := "PO1_2_REAL".Freon_11);
      NOP   0;
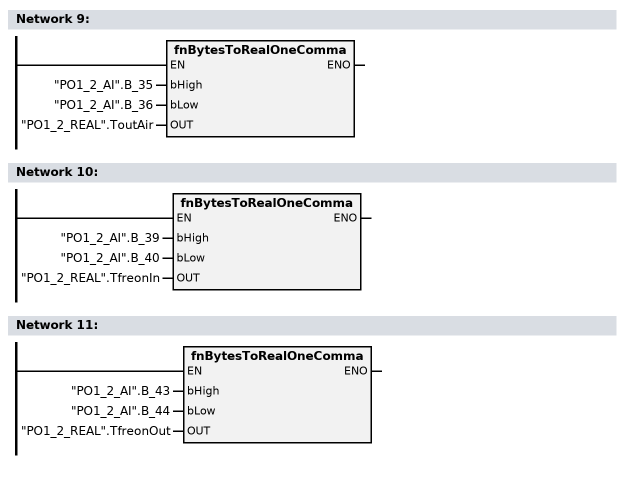
NETWORK
TITLE =
      CALL  "fnBytesToRealOneComma" (
           bHigh                    := "PO1_2_AI".B_35,
           bLow                     := "PO1_2_AI".B_36,
           OUT                      := "PO1_2_REAL".ToutAir);
      NOP   0;
NETWORK
TITLE =
      CALL  "fnBytesToRealOneComma" (
           bHigh                    := "PO1_2_AI".B_39,
           bLow                     := "PO1_2_AI".B_40,
           OUT                      := "PO1_2_REAL".TfreonIn);
      NOP   0;
NETWORK
TITLE =
      CALL  "fnBytesToRealOneComma" (
           bHigh                    := "PO1_2_AI".B_43,
           bLow                     := "PO1_2_AI".B_44,
           OUT                      := "PO1_2_REAL".TfreonOut);
      NOP   0;
END_FUNCTION_BLOCK

// FB 7: know-how protected block, not included

// FB 8: know-how protected block, not included

FUNCTION_BLOCK "GA1_1_GetReal"	// FB 9
VERSION : 0.1
BEGIN
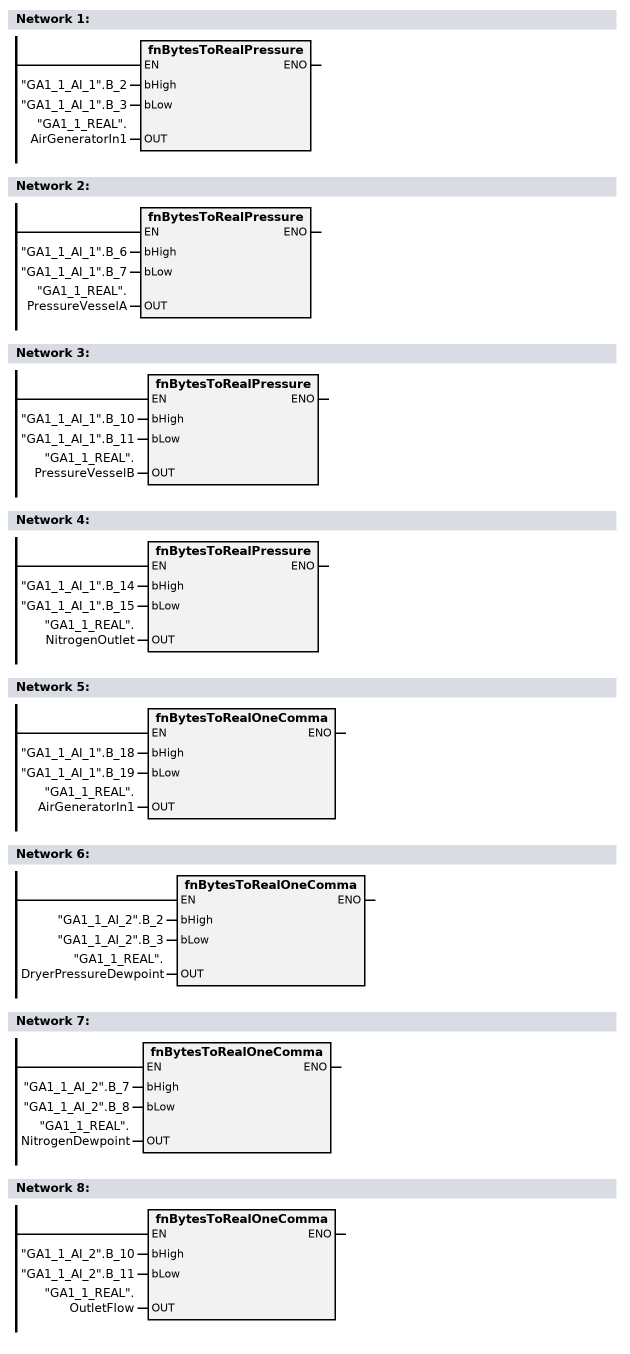
NETWORK
TITLE =
      CALL  "fnBytesToRealPressure" (
           bHigh                    := "GA1_1_AI_1".B_2,
           bLow                     := "GA1_1_AI_1".B_3,
           OUT                      := "GA1_1_REAL".AirGeneratorIn1);
      NOP   0;
NETWORK
TITLE =
      CALL  "fnBytesToRealPressure" (
           bHigh                    := "GA1_1_AI_1".B_6,
           bLow                     := "GA1_1_AI_1".B_7,
           OUT                      := "GA1_1_REAL".PressureVesselA);
      NOP   0;
NETWORK
TITLE =
      CALL  "fnBytesToRealPressure" (
           bHigh                    := "GA1_1_AI_1".B_10,
           bLow                     := "GA1_1_AI_1".B_11,
           OUT                      := "GA1_1_REAL".PressureVesselB);
      NOP   0;
NETWORK
TITLE =
      CALL  "fnBytesToRealPressure" (
           bHigh                    := "GA1_1_AI_1".B_14,
           bLow                     := "GA1_1_AI_1".B_15,
           OUT                      := "GA1_1_REAL".NitrogenOutlet);
      NOP   0;
NETWORK
TITLE =
      CALL  "fnBytesToRealOneComma" (
           bHigh                    := "GA1_1_AI_1".B_18,
           bLow                     := "GA1_1_AI_1".B_19,
           OUT                      := "GA1_1_REAL".AirGeneratorIn1);
      NOP   0;
NETWORK
TITLE =
      CALL  "fnBytesToRealOneComma" (
           bHigh                    := "GA1_1_AI_2".B_2,
           bLow                     := "GA1_1_AI_2".B_3,
           OUT                      := "GA1_1_REAL".DryerPressureDewpoint);
      NOP   0;
NETWORK
TITLE =
      CALL  "fnBytesToRealOneComma" (
           bHigh                    := "GA1_1_AI_2".B_7,
           bLow                     := "GA1_1_AI_2".B_8,
           OUT                      := "GA1_1_REAL".NitrogenDewpoint);
      NOP   0;
NETWORK
TITLE =
      CALL  "fnBytesToRealOneComma" (
           bHigh                    := "GA1_1_AI_2".B_10,
           bLow                     := "GA1_1_AI_2".B_11,
           OUT                      := "GA1_1_REAL".OutletFlow);
      NOP   0;
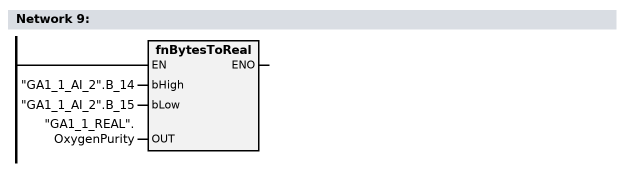
NETWORK
TITLE =
      CALL  "fnBytesToReal" (
           bHigh                    := "GA1_1_AI_2".B_14,
           bLow                     := "GA1_1_AI_2".B_15,
           OUT                      := "GA1_1_REAL".OxygenPurity);
      NOP   0;
END_FUNCTION_BLOCK

// FB 10: know-how protected block, not included

FUNCTION_BLOCK "GA1_2_GetReals"	// FB 11
VERSION : 0.1
BEGIN
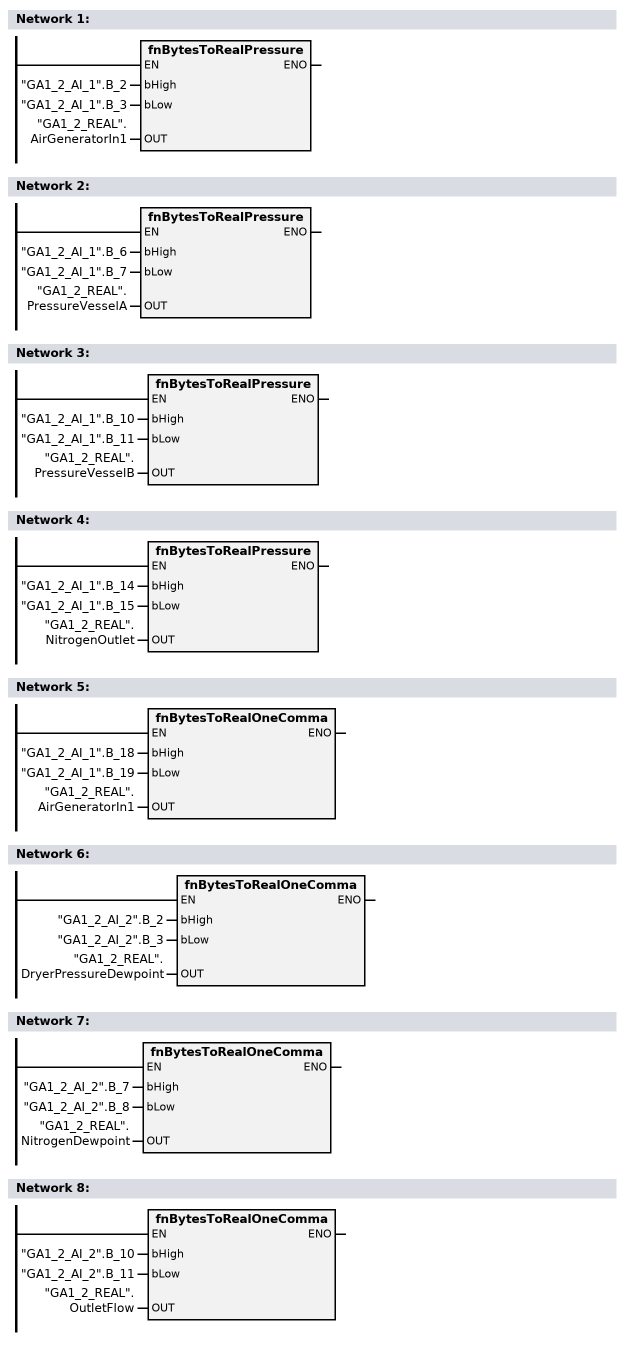
NETWORK
TITLE =
      CALL  "fnBytesToRealPressure" (
           bHigh                    := "GA1_2_AI_1".B_2,
           bLow                     := "GA1_2_AI_1".B_3,
           OUT                      := "GA1_2_REAL".AirGeneratorIn1);
      NOP   0;
NETWORK
TITLE =
      CALL  "fnBytesToRealPressure" (
           bHigh                    := "GA1_2_AI_1".B_6,
           bLow                     := "GA1_2_AI_1".B_7,
           OUT                      := "GA1_2_REAL".PressureVesselA);
      NOP   0;
NETWORK
TITLE =
      CALL  "fnBytesToRealPressure" (
           bHigh                    := "GA1_2_AI_1".B_10,
           bLow                     := "GA1_2_AI_1".B_11,
           OUT                      := "GA1_2_REAL".PressureVesselB);
      NOP   0;
NETWORK
TITLE =
      CALL  "fnBytesToRealPressure" (
           bHigh                    := "GA1_2_AI_1".B_14,
           bLow                     := "GA1_2_AI_1".B_15,
           OUT                      := "GA1_2_REAL".NitrogenOutlet);
      NOP   0;
NETWORK
TITLE =
      CALL  "fnBytesToRealOneComma" (
           bHigh                    := "GA1_2_AI_1".B_18,
           bLow                     := "GA1_2_AI_1".B_19,
           OUT                      := "GA1_2_REAL".AirGeneratorIn1);
      NOP   0;
NETWORK
TITLE =
      CALL  "fnBytesToRealOneComma" (
           bHigh                    := "GA1_2_AI_2".B_2,
           bLow                     := "GA1_2_AI_2".B_3,
           OUT                      := "GA1_2_REAL".DryerPressureDewpoint);
      NOP   0;
NETWORK
TITLE =
      CALL  "fnBytesToRealOneComma" (
           bHigh                    := "GA1_2_AI_2".B_7,
           bLow                     := "GA1_2_AI_2".B_8,
           OUT                      := "GA1_2_REAL".NitrogenDewpoint);
      NOP   0;
NETWORK
TITLE =
      CALL  "fnBytesToRealOneComma" (
           bHigh                    := "GA1_2_AI_2".B_10,
           bLow                     := "GA1_2_AI_2".B_11,
           OUT                      := "GA1_2_REAL".OutletFlow);
      NOP   0;
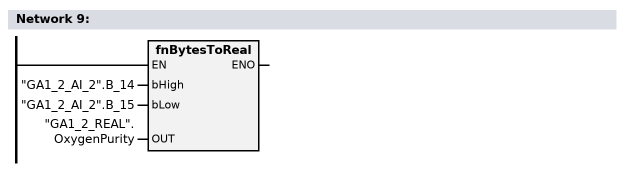
NETWORK
TITLE =
      CALL  "fnBytesToReal" (
           bHigh                    := "GA1_2_AI_2".B_14,
           bLow                     := "GA1_2_AI_2".B_15,
           OUT                      := "GA1_2_REAL".OxygenPurity);
      NOP   0;
END_FUNCTION_BLOCK

FUNCTION_BLOCK "GA2_1_GetReals"	// FB 12
VERSION : 0.1
BEGIN
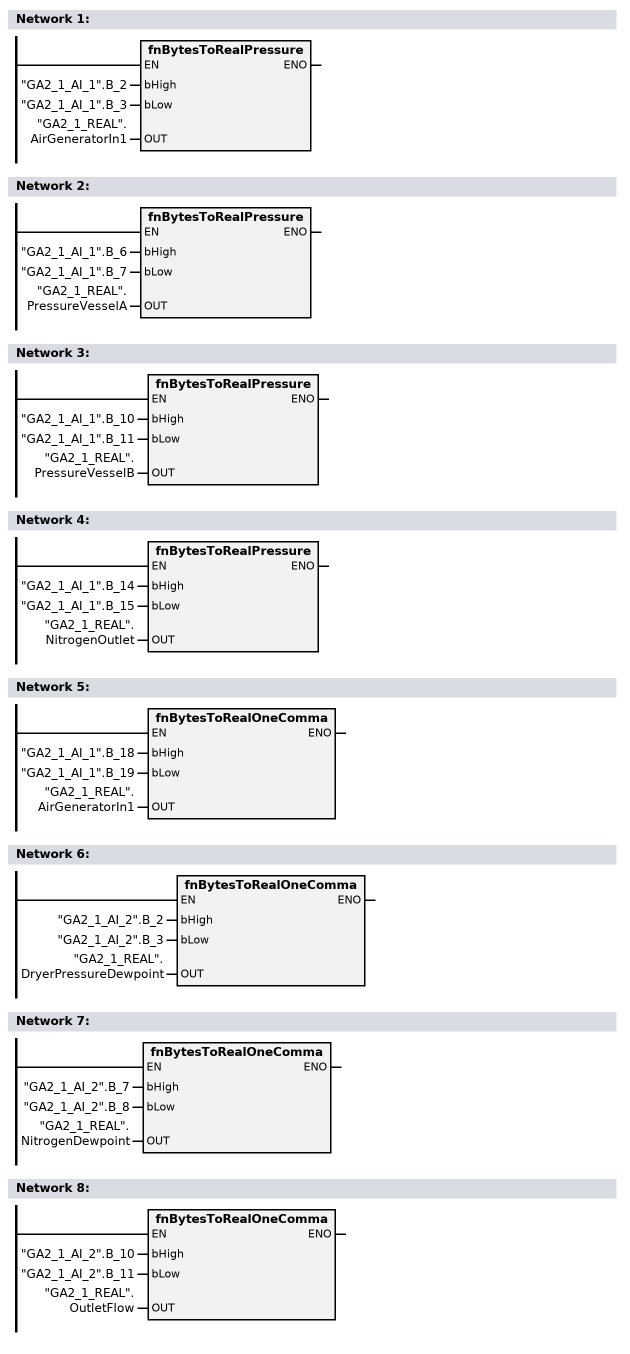
NETWORK
TITLE =
      CALL  "fnBytesToRealPressure" (
           bHigh                    := "GA2_1_AI_1".B_2,
           bLow                     := "GA2_1_AI_1".B_3,
           OUT                      := "GA2_1_REAL".AirGeneratorIn1);
      NOP   0;
NETWORK
TITLE =
      CALL  "fnBytesToRealPressure" (
           bHigh                    := "GA2_1_AI_1".B_6,
           bLow                     := "GA2_1_AI_1".B_7,
           OUT                      := "GA2_1_REAL".PressureVesselA);
      NOP   0;
NETWORK
TITLE =
      CALL  "fnBytesToRealPressure" (
           bHigh                    := "GA2_1_AI_1".B_10,
           bLow                     := "GA2_1_AI_1".B_11,
           OUT                      := "GA2_1_REAL".PressureVesselB);
      NOP   0;
NETWORK
TITLE =
      CALL  "fnBytesToRealPressure" (
           bHigh                    := "GA2_1_AI_1".B_14,
           bLow                     := "GA2_1_AI_1".B_15,
           OUT                      := "GA2_1_REAL".NitrogenOutlet);
      NOP   0;
NETWORK
TITLE =
      CALL  "fnBytesToRealOneComma" (
           bHigh                    := "GA2_1_AI_1".B_18,
           bLow                     := "GA2_1_AI_1".B_19,
           OUT                      := "GA2_1_REAL".AirGeneratorIn1);
      NOP   0;
NETWORK
TITLE =
      CALL  "fnBytesToRealOneComma" (
           bHigh                    := "GA2_1_AI_2".B_2,
           bLow                     := "GA2_1_AI_2".B_3,
           OUT                      := "GA2_1_REAL".DryerPressureDewpoint);
      NOP   0;
NETWORK
TITLE =
      CALL  "fnBytesToRealOneComma" (
           bHigh                    := "GA2_1_AI_2".B_7,
           bLow                     := "GA2_1_AI_2".B_8,
           OUT                      := "GA2_1_REAL".NitrogenDewpoint);
      NOP   0;
NETWORK
TITLE =
      CALL  "fnBytesToRealOneComma" (
           bHigh                    := "GA2_1_AI_2".B_10,
           bLow                     := "GA2_1_AI_2".B_11,
           OUT                      := "GA2_1_REAL".OutletFlow);
      NOP   0;
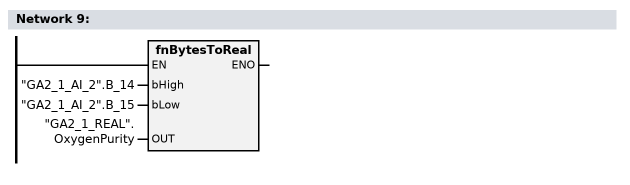
NETWORK
TITLE =
      CALL  "fnBytesToReal" (
           bHigh                    := "GA2_1_AI_2".B_14,
           bLow                     := "GA2_1_AI_2".B_15,
           OUT                      := "GA2_1_REAL".OxygenPurity);
      NOP   0;
END_FUNCTION_BLOCK

FUNCTION_BLOCK "GA2_2_GetReals"	// FB 13
VERSION : 0.1
BEGIN
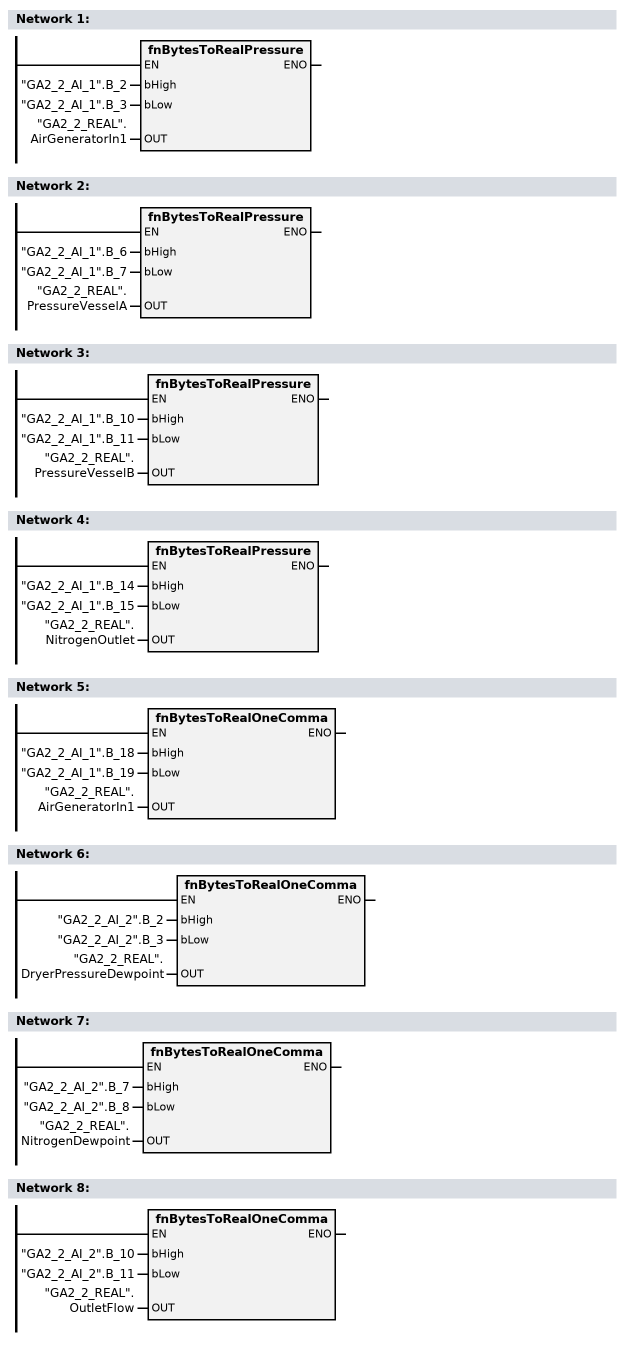
NETWORK
TITLE =
      CALL  "fnBytesToRealPressure" (
           bHigh                    := "GA2_2_AI_1".B_2,
           bLow                     := "GA2_2_AI_1".B_3,
           OUT                      := "GA2_2_REAL".AirGeneratorIn1);
      NOP   0;
NETWORK
TITLE =
      CALL  "fnBytesToRealPressure" (
           bHigh                    := "GA2_2_AI_1".B_6,
           bLow                     := "GA2_2_AI_1".B_7,
           OUT                      := "GA2_2_REAL".PressureVesselA);
      NOP   0;
NETWORK
TITLE =
      CALL  "fnBytesToRealPressure" (
           bHigh                    := "GA2_2_AI_1".B_10,
           bLow                     := "GA2_2_AI_1".B_11,
           OUT                      := "GA2_2_REAL".PressureVesselB);
      NOP   0;
NETWORK
TITLE =
      CALL  "fnBytesToRealPressure" (
           bHigh                    := "GA2_2_AI_1".B_14,
           bLow                     := "GA2_2_AI_1".B_15,
           OUT                      := "GA2_2_REAL".NitrogenOutlet);
      NOP   0;
NETWORK
TITLE =
      CALL  "fnBytesToRealOneComma" (
           bHigh                    := "GA2_2_AI_1".B_18,
           bLow                     := "GA2_2_AI_1".B_19,
           OUT                      := "GA2_2_REAL".AirGeneratorIn1);
      NOP   0;
NETWORK
TITLE =
      CALL  "fnBytesToRealOneComma" (
           bHigh                    := "GA2_2_AI_2".B_2,
           bLow                     := "GA2_2_AI_2".B_3,
           OUT                      := "GA2_2_REAL".DryerPressureDewpoint);
      NOP   0;
NETWORK
TITLE =
      CALL  "fnBytesToRealOneComma" (
           bHigh                    := "GA2_2_AI_2".B_7,
           bLow                     := "GA2_2_AI_2".B_8,
           OUT                      := "GA2_2_REAL".NitrogenDewpoint);
      NOP   0;
NETWORK
TITLE =
      CALL  "fnBytesToRealOneComma" (
           bHigh                    := "GA2_2_AI_2".B_10,
           bLow                     := "GA2_2_AI_2".B_11,
           OUT                      := "GA2_2_REAL".OutletFlow);
      NOP   0;
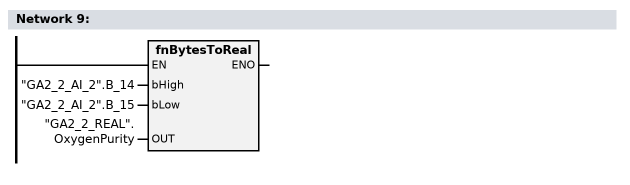
NETWORK
TITLE =
      CALL  "fnBytesToReal" (
           bHigh                    := "GA2_2_AI_2".B_14,
           bLow                     := "GA2_2_AI_2".B_15,
           OUT                      := "GA2_2_REAL".OxygenPurity);
      NOP   0;
END_FUNCTION_BLOCK

FUNCTION_BLOCK "KD_GetReals"	// FB 14
VERSION : 0.1
BEGIN
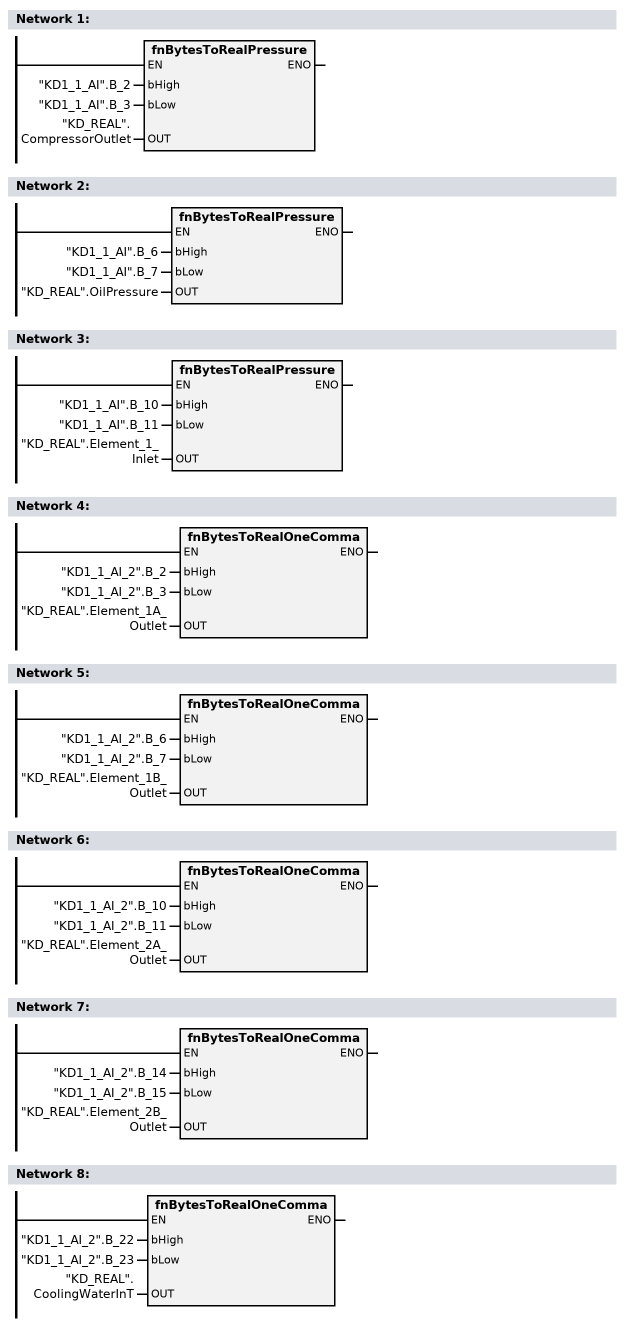
NETWORK
TITLE =
      CALL  "fnBytesToRealPressure" (
           bHigh                    := "KD1_1_AI".B_2,
           bLow                     := "KD1_1_AI".B_3,
           OUT                      := "KD_REAL".CompressorOutlet);
      NOP   0;
NETWORK
TITLE =
      CALL  "fnBytesToRealPressure" (
           bHigh                    := "KD1_1_AI".B_6,
           bLow                     := "KD1_1_AI".B_7,
           OUT                      := "KD_REAL".OilPressure);
      NOP   0;
NETWORK
TITLE =
      CALL  "fnBytesToRealPressure" (
           bHigh                    := "KD1_1_AI".B_10,
           bLow                     := "KD1_1_AI".B_11,
           OUT                      := "KD_REAL".Element_1_Inlet);
      NOP   0;
NETWORK
TITLE =
      CALL  "fnBytesToRealOneComma" (
           bHigh                    := "KD1_1_AI_2".B_2,
           bLow                     := "KD1_1_AI_2".B_3,
           OUT                      := "KD_REAL".Element_1A_Outlet);
      NOP   0;
NETWORK
TITLE =
      CALL  "fnBytesToRealOneComma" (
           bHigh                    := "KD1_1_AI_2".B_6,
           bLow                     := "KD1_1_AI_2".B_7,
           OUT                      := "KD_REAL".Element_1B_Outlet);
      NOP   0;
NETWORK
TITLE =
      CALL  "fnBytesToRealOneComma" (
           bHigh                    := "KD1_1_AI_2".B_10,
           bLow                     := "KD1_1_AI_2".B_11,
           OUT                      := "KD_REAL".Element_2A_Outlet);
      NOP   0;
NETWORK
TITLE =
      CALL  "fnBytesToRealOneComma" (
           bHigh                    := "KD1_1_AI_2".B_14,
           bLow                     := "KD1_1_AI_2".B_15,
           OUT                      := "KD_REAL".Element_2B_Outlet);
      NOP   0;
NETWORK
TITLE =
      CALL  "fnBytesToRealOneComma" (
           bHigh                    := "KD1_1_AI_2".B_22,
           bLow                     := "KD1_1_AI_2".B_23,
           OUT                      := "KD_REAL".CoolingWaterInT);
      NOP   0;
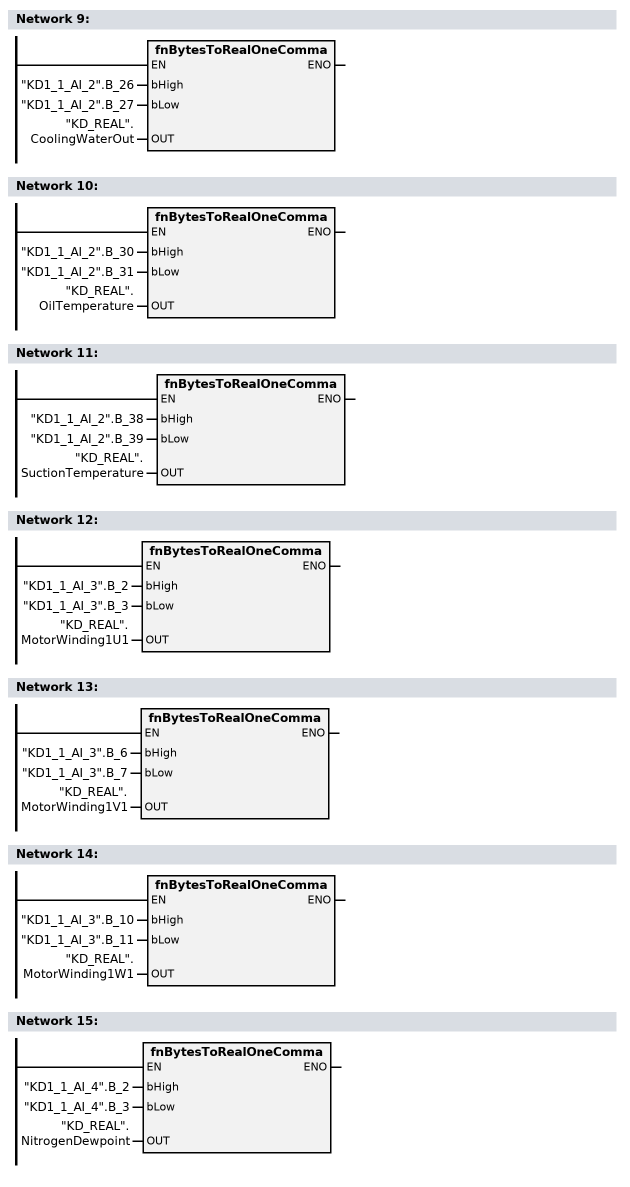
NETWORK
TITLE =
      CALL  "fnBytesToRealOneComma" (
           bHigh                    := "KD1_1_AI_2".B_26,
           bLow                     := "KD1_1_AI_2".B_27,
           OUT                      := "KD_REAL".CoolingWaterOut);
      NOP   0;
NETWORK
TITLE =
      CALL  "fnBytesToRealOneComma" (
           bHigh                    := "KD1_1_AI_2".B_30,
           bLow                     := "KD1_1_AI_2".B_31,
           OUT                      := "KD_REAL".OilTemperature);
      NOP   0;
NETWORK
TITLE =
      CALL  "fnBytesToRealOneComma" (
           bHigh                    := "KD1_1_AI_2".B_38,
           bLow                     := "KD1_1_AI_2".B_39,
           OUT                      := "KD_REAL".SuctionTemperature);
      NOP   0;
NETWORK
TITLE =
      CALL  "fnBytesToRealOneComma" (
           bHigh                    := "KD1_1_AI_3".B_2,
           bLow                     := "KD1_1_AI_3".B_3,
           OUT                      := "KD_REAL".MotorWinding1U1);
      NOP   0;
NETWORK
TITLE =
      CALL  "fnBytesToRealOneComma" (
           bHigh                    := "KD1_1_AI_3".B_6,
           bLow                     := "KD1_1_AI_3".B_7,
           OUT                      := "KD_REAL".MotorWinding1V1);
      NOP   0;
NETWORK
TITLE =
      CALL  "fnBytesToRealOneComma" (
           bHigh                    := "KD1_1_AI_3".B_10,
           bLow                     := "KD1_1_AI_3".B_11,
           OUT                      := "KD_REAL".MotorWinding1W1);
      NOP   0;
NETWORK
TITLE =
      CALL  "fnBytesToRealOneComma" (
           bHigh                    := "KD1_1_AI_4".B_2,
           bLow                     := "KD1_1_AI_4".B_3,
           OUT                      := "KD_REAL".NitrogenDewpoint);
      NOP   0;
END_FUNCTION_BLOCK

FUNCTION_BLOCK "ModbusReal"	// FB 15
VERSION : 0.1
BEGIN
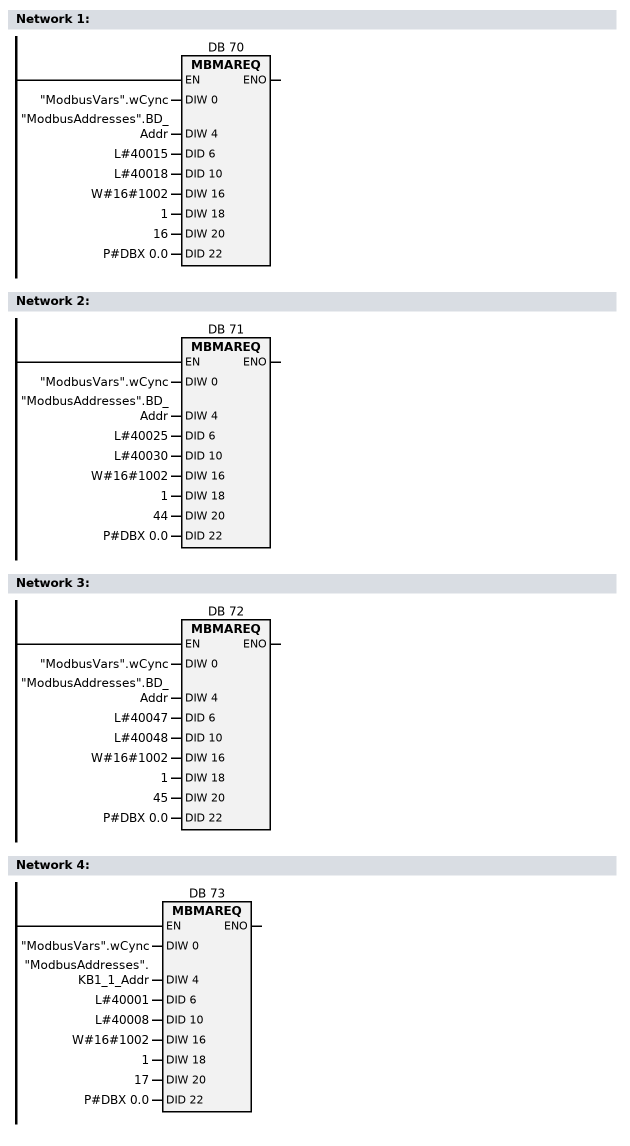
NETWORK
TITLE =
      CALL  "MBMAREQ" , DB 70 (
           DIW 0                    := "ModbusVars".wCync,
           DIW 4                    := "ModbusAddresses".BD_Addr,
           DID 6                    := L#40015,
           DID 10                   := L#40018,
           DIW 16                   := W#16#1002,
           DIW 18                   := 1,
           DIW 20                   := 16,
           DID 22                   := P#DBX 0.0);
      NOP   0;
NETWORK
TITLE =
      CALL  "MBMAREQ" , DB 71 (
           DIW 0                    := "ModbusVars".wCync,
           DIW 4                    := "ModbusAddresses".BD_Addr,
           DID 6                    := L#40025,
           DID 10                   := L#40030,
           DIW 16                   := W#16#1002,
           DIW 18                   := 1,
           DIW 20                   := 44,
           DID 22                   := P#DBX 0.0);
      NOP   0;
NETWORK
TITLE =
      CALL  "MBMAREQ" , DB 72 (
           DIW 0                    := "ModbusVars".wCync,
           DIW 4                    := "ModbusAddresses".BD_Addr,
           DID 6                    := L#40047,
           DID 10                   := L#40048,
           DIW 16                   := W#16#1002,
           DIW 18                   := 1,
           DIW 20                   := 45,
           DID 22                   := P#DBX 0.0);
      NOP   0;
NETWORK
TITLE =
      CALL  "MBMAREQ" , DB 73 (
           DIW 0                    := "ModbusVars".wCync,
           DIW 4                    := "ModbusAddresses".KB1_1_Addr,
           DID 6                    := L#40001,
           DID 10                   := L#40008,
           DIW 16                   := W#16#1002,
           DIW 18                   := 1,
           DIW 20                   := 17,
           DID 22                   := P#DBX 0.0);
      NOP   0;
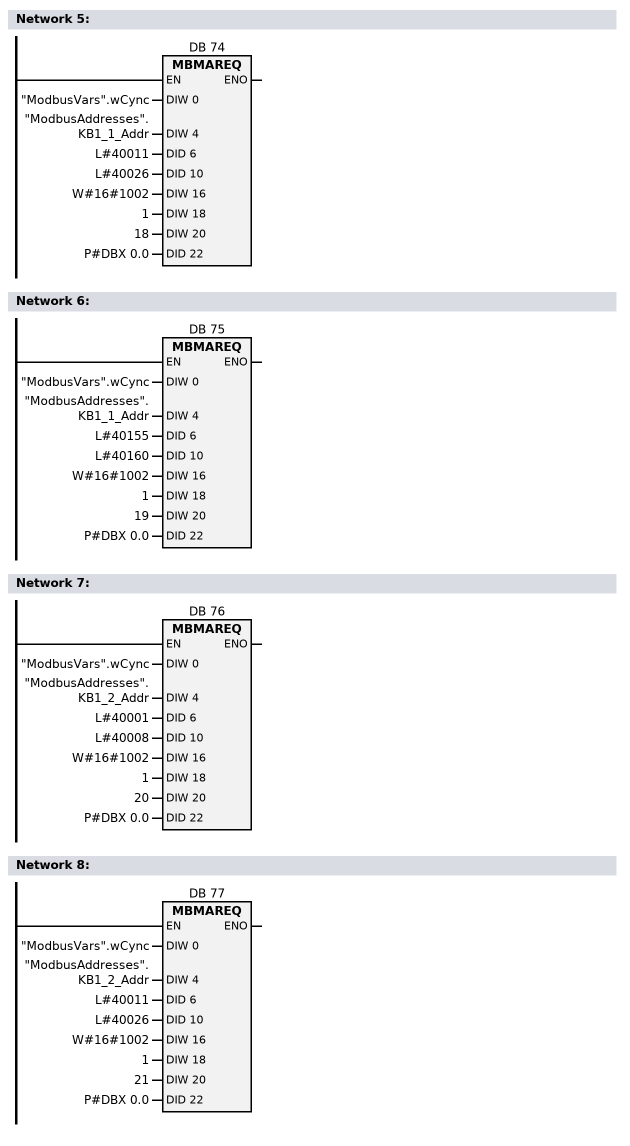
NETWORK
TITLE =
      CALL  "MBMAREQ" , DB 74 (
           DIW 0                    := "ModbusVars".wCync,
           DIW 4                    := "ModbusAddresses".KB1_1_Addr,
           DID 6                    := L#40011,
           DID 10                   := L#40026,
           DIW 16                   := W#16#1002,
           DIW 18                   := 1,
           DIW 20                   := 18,
           DID 22                   := P#DBX 0.0);
      NOP   0;
NETWORK
TITLE =
      CALL  "MBMAREQ" , DB 75 (
           DIW 0                    := "ModbusVars".wCync,
           DIW 4                    := "ModbusAddresses".KB1_1_Addr,
           DID 6                    := L#40155,
           DID 10                   := L#40160,
           DIW 16                   := W#16#1002,
           DIW 18                   := 1,
           DIW 20                   := 19,
           DID 22                   := P#DBX 0.0);
      NOP   0;
NETWORK
TITLE =
      CALL  "MBMAREQ" , DB 76 (
           DIW 0                    := "ModbusVars".wCync,
           DIW 4                    := "ModbusAddresses".KB1_2_Addr,
           DID 6                    := L#40001,
           DID 10                   := L#40008,
           DIW 16                   := W#16#1002,
           DIW 18                   := 1,
           DIW 20                   := 20,
           DID 22                   := P#DBX 0.0);
      NOP   0;
NETWORK
TITLE =
      CALL  "MBMAREQ" , DB 77 (
           DIW 0                    := "ModbusVars".wCync,
           DIW 4                    := "ModbusAddresses".KB1_2_Addr,
           DID 6                    := L#40011,
           DID 10                   := L#40026,
           DIW 16                   := W#16#1002,
           DIW 18                   := 1,
           DIW 20                   := 21,
           DID 22                   := P#DBX 0.0);
      NOP   0;
